(* IEC 61131-3 sources: volt/packages/volt-lsp-iec/test-corpus/pro2193/Device/Plc Logic/Application/09 Misc/Library Manager/L_MC1P_MotionControlBasic (part 5) *)

(* ---- L_MC1P_MOTIONUTILS_I750.pou ---- *)
FUNCTION_BLOCK L_MC1P_MOTIONUTILS_I750 EXTENDS L_MC1P_MotionUtils_Base
VAR
	DRIVETYPE : L_MC1P_DriveType;
	GETAXISEXTENSION : L_MC1P_AxisExtensionTypes;
END_VAR
END_FUNCTION_BLOCK

METHOD GETRETAINMEMINFO : L_MC1P_RetainDataType
VAR_OUTPUT
	MEMINFO : L_MC1P_uAxisRetainInfo;
END_VAR
END_METHOD

(* ---- L_MC1P_MOTIONUTILS_I950.pou ---- *)
FUNCTION_BLOCK L_MC1P_MOTIONUTILS_I950 EXTENDS L_MC1P_MotionUtils_Base
VAR
	DRIVETYPE : L_MC1P_DriveType;
	GETAXISEXTENSION : L_MC1P_AxisExtensionTypes;
END_VAR
END_FUNCTION_BLOCK

METHOD GETRETAINMEMINFO : L_MC1P_RetainDataType
VAR_OUTPUT
	MEMINFO : L_MC1P_uAxisRetainInfo;
END_VAR
END_METHOD

(* ---- L_MC1P_MOTIONUTILS_I950_CIAADV.pou ---- *)
FUNCTION_BLOCK L_MC1P_MOTIONUTILS_I950_CIAADV EXTENDS L_MC1P_MotionUtils_Base
VAR
	DRIVETYPE : L_MC1P_DriveType;
	GETAXISEXTENSION : L_MC1P_AxisExtensionTypes;
END_VAR
END_FUNCTION_BLOCK

METHOD GETRETAINMEMINFO : L_MC1P_RetainDataType
VAR_OUTPUT
	MEMINFO : L_MC1P_uAxisRetainInfo;
END_VAR
END_METHOD

(* ---- L_MC1P_MOTIONUTILS_I950_DRIVE.pou ---- *)
FUNCTION_BLOCK L_MC1P_MOTIONUTILS_I950_DRIVE EXTENDS L_MC1P_MotionUtils_Base
VAR
	DRIVETYPE : L_MC1P_DriveType;
	GETAXISEXTENSION : L_MC1P_AxisExtensionTypes;
END_VAR
END_FUNCTION_BLOCK

METHOD GETGUID : BOOL
VAR_INPUT
	PCONNECTOR : POINTER TO IoConfigConnector;
END_VAR
VAR_IN_OUT
	GUID : L_MC1P_AxisGUID;
END_VAR
END_METHOD

METHOD GETRETAINMEMINFO : L_MC1P_RetainDataType
VAR_OUTPUT
	MEMINFO : L_MC1P_uAxisRetainInfo;
END_VAR
END_METHOD

(* ---- L_MC1P_MOTIONUTILSRETAINHANDLING.pou ---- *)
FUNCTION_BLOCK L_MC1P_MOTIONUTILSRETAINHANDLING
VAR_INPUT
	XRETAINSTART : BOOL;
END_VAR
VAR
	PAXISREAL : POINTER TO _AXIS_REF_REAL;
	PAXISRETAININFORMATION : POINTER TO L_MC1P_AxisRetainInformation;
	RETAININFO : L_MC1P_uAxisRetainInfo;
	ERETAINDATATYPE : L_MC1P_RetainDataType := L_MC1P_RetainDataType.DataRealDrive;
	PRETAINDATA : POINTER TO L_MC1P_uRetainData;
	UINITIALRETAINDATA : L_MC1P_uRetainData;
	XERR_XPOSRECONSTRDATAVERSIONCHANGED : BOOL;
	XERR_POSRECONSTRNODATAAVAILABLE : BOOL;
	XRETAINDATAAVAILABLE : BOOL;
	WRETAINERRORSTATE : WORD;
	WRETAINSTATE : WORD;
	CHECKDRIVEGUID : BOOL;
	DRIVEGUID : L_MC1P_AxisGUID;
	GETAXIS : POINTER TO _Axis_Ref_Real;
	INFO : DWORD;
	ITFRETAINFUNCTION : L_MC1P_IRetainFunction;
	RETAINDATAAVAILABLE : BOOL;
	RETAINDATACONFIGURED : BOOL;
	RETAINSTATE : WORD;
END_VAR
END_FUNCTION_BLOCK

METHOD COPYRETAINDATABYVERSION : BOOL
VAR_INPUT
	PDATA : POINTER TO DWORD;
	INFO : DWORD;
END_VAR
END_METHOD

METHOD GETINITIALDATA : BOOL
VAR_INPUT
	PDATA : POINTER TO DWORD;
	INFO : DWORD;
END_VAR
END_METHOD

METHOD GETINITIALRETAINDATA : POINTER TO L_MC1P_uRetainData
VAR_INPUT
	XNEWEST : BOOL;
END_VAR
END_METHOD

METHOD GETRETAINSTATE : WORD
VAR_OUTPUT
	WSTATERETAINERROR : WORD;
END_VAR
END_METHOD

METHOD REGISTERONRETAINDATAHANDLER
VAR_INPUT
	AXISGUID : L_MC1P_AxisGUID;
END_VAR
END_METHOD

METHOD RESET
END_METHOD

METHOD SETCONNECTEDGUID : BOOL
VAR_INPUT
	GUID : L_MC1P_AxisGUID;
END_VAR
END_METHOD

METHOD SETERRORINFO
VAR_INPUT
	WSTATE : WORD;
END_VAR
END_METHOD

METHOD SETINITIALDATA : BOOL
VAR_INPUT
	PDATA : POINTER TO DWORD;
END_VAR
END_METHOD

METHOD STOREDATA
VAR_INPUT
	PDATA : POINTER TO DWORD;
END_VAR
END_METHOD

METHOD FB_INIT : BOOL
VAR_INPUT
	BINITRETAINS : BOOL;
	BINCOPYCODE : BOOL;
	MEMLENGTH : WORD;
	MEMTYPE : BYTE;
	MEMVERSION : BYTE;
	ERETAINDATATYPE : L_MC1P_RetainDataType;
END_VAR
END_METHOD

(* ---- L_MC1P_MOTIONUTILSRETAINHANDLINGEXTFB.pou ---- *)
FUNCTION_BLOCK L_MC1P_MOTIONUTILSRETAINHANDLINGEXTFB
VAR_INPUT
	XRETAINDATAAVAILABLE : BOOL;
	PRETAINDATA : POINTER TO L_MC1P_uRetainData;
	WRETAINSTATE : WORD;
END_VAR
VAR
	CHECKDRIVEGUID : BOOL;
	DRIVEGUID : L_MC1P_AxisGUID;
	GETAXIS : POINTER TO _Axis_Ref_Real;
	ITFRETAINFUNCTION : L_MC1P_IRetainFunction;
	RETAINDATAAVAILABLE : BOOL;
END_VAR
END_FUNCTION_BLOCK

METHOD GETINITIALRETAINDATA : POINTER TO L_MC1P_uRetainData
VAR_INPUT
	XNEWEST : BOOL;
END_VAR
END_METHOD

METHOD GETRETAINSTATE : WORD
VAR_OUTPUT
	WSTATERETAINERROR : WORD;
END_VAR
END_METHOD

METHOD REGISTERONRETAINDATAHANDLER
VAR_INPUT
	AXISGUID : L_MC1P_AxisGUID;
END_VAR
END_METHOD

METHOD RESET
END_METHOD

METHOD SETCONNECTEDGUID : BOOL
VAR_INPUT
	GUID : L_MC1P_AxisGUID;
END_VAR
END_METHOD

(* ---- L_MC1P_MOTIONUTILSRETAINHANDLINGUNIVERSAL.pou ---- *)
FUNCTION_BLOCK L_MC1P_MOTIONUTILSRETAINHANDLINGUNIVERSAL EXTENDS L_MC1P_MotionUtilsRetainHandling
VAR
	MYDRIVEGUID : L_MC1P_AxisGUID;
	CHECKDRIVEGUID : BOOL;
	DRIVEGUID : L_MC1P_AxisGUID;
END_VAR
END_FUNCTION_BLOCK

METHOD GETINITIALRETAINDATA : POINTER TO L_MC1P_uRetainData
VAR_INPUT
	XNEWEST : BOOL;
END_VAR
END_METHOD

METHOD RESET
END_METHOD

METHOD SETCONNECTEDGUID : BOOL
VAR_INPUT
	GUID : L_MC1P_AxisGUID;
END_VAR
END_METHOD

METHOD STOREDATA
VAR_INPUT
	PDATA : POINTER TO DWORD;
END_VAR
END_METHOD

(* ---- L_MC1P_MOVEABSOLUTE_INERNAL.pou ---- *)
FUNCTION_BLOCK L_MC1P_MOVEABSOLUTE_INERNAL EXTENDS L_MC1P_Template_IntFB
VAR_INPUT
	EXECUTE : BOOL;
	CONTINUOUSUPDATE : BOOL;
	POSITION : LREAL;
	VELOCITY : LREAL;
	ACCELERATION : LREAL;
	DECELERATION : LREAL;
	JERK : LREAL;
	JERKDEC : LREAL;
	DIRECTION : MC_DIRECTION;
	BUFFERMODE : MC_BUFFER_MODE;
END_VAR
VAR_OUTPUT
	DONE : BOOL;
	BUSY : BOOL;
	ACTIVE : BOOL;
	COMMANDABORTED : BOOL;
	ERROR : BOOL;
	ERRORID : L_IE1P_Error;
END_VAR
VAR
	FBMB : L_MC1P_MoveBasic := STRUCT(wCalcProfileMode := 1);
	XUSED : BOOL;
	ABORTEDBYLIMIT : BOOL;
END_VAR
END_FUNCTION_BLOCK

METHOD MAIN
VAR_IN_OUT
	AXIS : AXIS_REF;
	FBBASE : L_MC1P_Template_ForAxis;
END_VAR
END_METHOD

(* ---- L_MC1P_MOVEBASIC.pou ---- *)
FUNCTION_BLOCK L_MC1P_MOVEBASIC
VAR_INPUT
	LRJERKDEC : LREAL := 0;
	XWAIT : BOOL;
	XRECALCULATE : BOOL;
	LRCORRECTTIMEBASE : LREAL;
	WCALCPROFILEMODE : WORD := 0;
	XUSEEXTERNPROFILECALCULATION : BOOL;
	ITFPOSPROFILECALCULATION : L_MC1P_IPosProfileCalculation;
	XENABLEOFFSETVELOCITY : BOOL;
	LROFFSETVELOCITY : LREAL;
	XFINISHPOSFROMMOVEREL : BOOL := FALSE;
END_VAR
VAR
	XSTART : BOOL;
	EXECUTEOLD : BOOL;
	COMMANDABORTEDOLD : BOOL;
	PG : REFERENCE TO L_MC1P_PosProfiler;
	SCPARAM : L_MC1P_ProfileParameter;
	SCPARAMLIM : L_MC1P_ProfileParameter;
	WFUNID : WORD;
	XSETENDVELOCITYBYBUFFERMODE : BOOL;
	XRESETOUTPUT : BOOL;
	EACTSTATE : L_MC1P_AXIS_STATE;
	XCONTINUOUSUPDATEACTIVE : BOOL;
	XSUPERIMPOSED : BOOL;
	XPOSACTIVE : BOOL;
	XVELUPDATE : BOOL;
	XBUFFERACTIVE : BOOL;
	XPOSSWLIMIT : BOOL;
	XNEGSWLIMIT : BOOL;
	XABORTEDBYLIMIT : BOOL;
	XWARNING : BOOL;
	EWARNINGID : L_IE1P_Error;
	XWARNINGOLD : BOOL;
	EWARNINGIDOLD : L_IE1P_Error;
	XLOGINFO : BOOL;
	ELOGINFOID : L_IE1P_Error;
	ELOGINFOIDOLD : L_IE1P_Error;
	XLIMITOLD : BOOL;
	XCONTMODE : BOOL;
	XDONESAVE : BOOL;
	LRPOSLATCHED : LREAL;
	LRPOSSAVE : LREAL;
	XDONEOLD : BOOL;
	LRDISTANCE : LREAL;
	LRSTARTPOS : LREAL;
	LRTMPPOSOFFSET : LREAL;
	XIGNOREMODULOWINDOW : BOOL;
	SCPROFILEDATATMP : L_MC1P_ProfileData;
	SCPROFILEPARATMP : L_MC1P_ProfileParameter;
	XNEWPROFILESTARTAFTERSTANDSTILL : BOOL;
	ESETDIRECTIONMOVEFB : MC_DIRECTION;
	XPOSPROFILERINUSE : BOOL;
	WSTRETCHPROFILEMODE : WORD;
	XBUFFERDATAUPDATED : BOOL;
	XENABLEBUFFER_INT : BOOL;
	SCBUFFERDATA_INT : L_MC1P_BufferData;
	XUPDATEBUFFERDATAFROMDUMMYPG : BOOL;
	PAXIS : POINTER TO AXIS_REF;
	IGNOREMODULOWINDOW : BOOL;
	POSPROFILERINUSE : BOOL;
	PROFILETIME : TIME;
	REMAININGTIMEOFPROFILE : LREAL;
	REMAININGTIMEOFPROFILEAVAILABLE : BOOL;
	STRETCHPROFILEMODE : WORD;
END_VAR
END_FUNCTION_BLOCK

METHOD CALCTARGETPOSITION : LREAL
VAR_INPUT
	POSITION : LREAL;
	DIRECTION : MC_DIRECTION;
	ETRAVERSINGRANGE : L_MC1P_TraversingRange;
	ETYPEFUNCTION : L_MC1P_TypeFunction;
	XFIRSTCALC : BOOL;
	XABORTED : BOOL;
	PROFILEPARAM : L_MC1P_ProfileParameter;
	EAXISSTATEOLD : L_MC1P_AXIS_STATE;
END_VAR
VAR_OUTPUT
	XERROR : BOOL;
	EERRORID : L_IE1P.L_IE1P_Error;
END_VAR
VAR_IN_OUT
	AXIS : AXIS_REF;
END_VAR
END_METHOD

METHOD CHECKDEVIATION : BOOL
VAR_INPUT
	LRINPUT : LREAL;
	LRSAVE : LREAL;
END_VAR
END_METHOD

METHOD CHECKLIMITATION
VAR_INPUT
	EFUNCTIONTYP : L_MC1P_TypeFunction;
	PXPOSMODE : POINTER TO BOOL;
END_VAR
VAR_IN_OUT
	AXIS : AXIS_REF;
	FBBASE : L_MC1P_Template_ForAxis;
	ERROR : BOOL;
	ERRORID : L_IE1P_Error;
END_VAR
END_METHOD

METHOD DETERMINETARGETSPEEDSIGN : BOOL
VAR_INPUT
	LRPOSITION : LREAL;
	ETYPEFUNCTION : L_MC1P_TypeFunction;
	EDIRECTION : MC_DIRECTION;
END_VAR
VAR_IN_OUT
	AXIS : AXIS_REF;
END_VAR
END_METHOD

METHOD INTOLERANCEWINDOW : BOOL
VAR_INPUT
	LRPOSITION : LREAL;
END_VAR
VAR_OUTPUT
	DIRECTION : MC_DIRECTION;
END_VAR
VAR_IN_OUT
	AXIS : AXIS_REF;
END_VAR
END_METHOD

METHOD PREPAREBUFFERDATA
VAR_INPUT
	XENABLEBUFFER : BOOL;
	SCBUFFERDATA : L_MC1P_BufferData;
END_VAR
END_METHOD

METHOD PROFILER : BOOL
VAR_INPUT
	EXECUTE : BOOL;
	CONTINUOUSUPDATE : BOOL;
	POSITION : LREAL;
	VELOCITY : LREAL;
	ENDVELOCITY : LREAL;
	ACCELERATION : LREAL;
	DECELERATION : LREAL;
	JERK : LREAL;
	XPOSMODE : BOOL;
	DIRECTION : MC_DIRECTION;
	BUFFERMODE : MC_BUFFER_MODE;
	EFUNCTIONTYP : L_MC1P_TypeFunction;
END_VAR
VAR_IN_OUT
	AXIS : AXIS_REF;
	DONE : BOOL;
	BUSY : BOOL;
	ACTIVE : BOOL;
	COMMANDABORTED : BOOL;
	ERROR : BOOL;
	ERRORID : L_IE1P_Error;
	FBBASE : L_MC1P_Template_ForAxis;
END_VAR
END_METHOD

METHOD RESET
END_METHOD

METHOD RESETEXECUTE
END_METHOD

(* ---- L_MC1P_MOVERELATIVE_INTERNAL.pou ---- *)
FUNCTION_BLOCK L_MC1P_MOVERELATIVE_INTERNAL EXTENDS L_MC1P_Template_IntFB
VAR_INPUT
	EXECUTE : BOOL;
	CONTINUOUSUPDATE : BOOL;
	DISTANCE : LREAL;
	VELOCITY : LREAL;
	ACCELERATION : LREAL;
	DECELERATION : LREAL;
	JERK : LREAL;
	JERKDEC : LREAL;
	BUFFERMODE : MC_BUFFER_MODE;
	XUSEEXTERNPROFILECALCULATION : BOOL;
	ITFPOSPROFILECALCULATION : L_MC1P_IPosProfileCalculation;
END_VAR
VAR_OUTPUT
	DONE : BOOL;
	BUSY : BOOL;
	ACTIVE : BOOL;
	COMMANDABORTED : BOOL;
	ERROR : BOOL;
	ERRORID : L_IE1P_Error;
END_VAR
VAR
	FBMB : L_MC1P_MoveBasic := STRUCT(wCalcProfileMode := 1);
	XUSED : BOOL;
	ABORTEDBYLIMIT : BOOL;
END_VAR
END_FUNCTION_BLOCK

METHOD MAIN
VAR_IN_OUT
	AXIS : AXIS_REF;
	FBBASE : L_MC1P_Template_ForAxis;
END_VAR
END_METHOD

(* ---- L_MC1P_MOVEVELOCITY_INTERNAL.pou ---- *)
FUNCTION_BLOCK L_MC1P_MOVEVELOCITY_INTERNAL EXTENDS L_MC1P_Template_IntFB
VAR_INPUT
	EXECUTE : BOOL;
	CONTINUOUSUPDATE : BOOL;
	VELOCITY : LREAL;
	ACCELERATION : LREAL;
	DECELERATION : LREAL;
	JERK : LREAL;
	JERKDEC : LREAL;
	DIRECTION : MC_DIRECTION := MC_DIRECTION.mcPositiveDirection;
	BUFFERMODE : MC_BUFFER_MODE;
	XUSEEXTERNPROFILECALCULATION : BOOL;
	ITFPOSPROFILECALCULATION : L_MC1P_IPosProfileCalculation;
	XENABLEOFFSETVELOCITY : BOOL;
	LROFFSETVELOCITY : LREAL;
END_VAR
VAR_OUTPUT
	INVELOCITY : BOOL;
	BUSY : BOOL;
	ACTIVE : BOOL;
	COMMANDABORTED : BOOL;
	ERROR : BOOL;
	ERRORID : L_IE1P_Error;
END_VAR
VAR
	FBMB : L_MC1P_MoveBasic := STRUCT(wCalcProfileMode := 1);
	LRVEL : LREAL;
	XUSED : BOOL;
	ABORTEDBYLIMIT : BOOL;
END_VAR
END_FUNCTION_BLOCK

METHOD MAIN
VAR_IN_OUT
	AXIS : AXIS_REF;
	FBBASE : L_MC1P_Template_ForAxis;
END_VAR
END_METHOD

METHOD MODVELOCITY : LREAL
VAR_IN_OUT
	AXIS : AXIS_REF;
END_VAR
END_METHOD

(* ---- L_MC1P_MPOT.pou ---- *)
FUNCTION_BLOCK L_MC1P_MPOT
VAR_INPUT
	XENABLE : BOOL;
	XJOGPOS : BOOL;
	XJOGNEG : BOOL;
	LRVELPOS : LREAL;
	LRVELNEG : LREAL;
	LRACC : LREAL;
	LRDEC : LREAL;
	LRDECDISABLE : LREAL;
END_VAR
VAR_OUTPUT
	XBUSY : BOOL;
	LRSETVELOUT : LREAL;
END_VAR
VAR
	HLP_MPOT : L_MC1P_HlpRampGenerator;
	XJOGPOSITIVEFLAG : BOOL;
	XJOGNEGATIVEFLAG : BOOL;
END_VAR
END_FUNCTION_BLOCK

(* ---- L_MC1P_NOISEDETECTION.pou ---- *)
FUNCTION_BLOCK L_MC1P_NOISEDETECTION
VAR_INPUT
	XENABLE : BOOL;
	LRCYCPOS : LREAL;
	LRCYCVEL : LREAL;
	LRCYCACC : LREAL;
	ECYCVALUEMODE : L_MC1P_SetValueMode := L_MC1P_SetValueMode.Vel;
	LRCYCLELENGTH : LREAL := 360;
	ETRAVERSINGRANGE : L_MC1P_TraversingRange;
END_VAR
VAR_OUTPUT
	XBUSY : BOOL;
	XNOISEDETECTED : BOOL;
END_VAR
VAR
	WSTATE : WORD;
	XNOISE_INT : BOOL;
	LRDELTAPOS_INT : LREAL;
	WNOISEDETECTEDCOUNT : WORD;
	WNOISENOTDETECTEDCOUNT : WORD;
	XENABLE_OLD : BOOL;
	LRCYCPOS_OLD : LREAL;
	LRCYCVEL_OLD : LREAL;
	LRDELTAPOS_OLD : LREAL;
	FB_STACK : L_MC1P_StackControlArray := STRUCT(iMaxLegth := ciArraylengthAtCheckNoise);
	ALRACC : ARRAY [1..ciArraylengthAtCheckNoise] OF LREAL;
	ALRDELTA2POS : ARRAY [1..ciArraylengthAtCheckNoise] OF LREAL;
	ALRDELTAVEL : ARRAY [1..ciArraylengthAtCheckNoise] OF LREAL;
	CIARRAYLENGTHATCHECKNOISE : INT := 15;
	C_WHYSTCOUNTERNOISEDETECTED : WORD := 3;
END_VAR
END_FUNCTION_BLOCK

METHOD CALL_ERRORHANDLER
END_METHOD

METHOD CALL_FBMETHODS
END_METHOD

METHOD CALL_OUTPUT
END_METHOD

METHOD CALL_RESETCOMMANDS
END_METHOD

METHOD CALL_RESETOUTPUT
END_METHOD

METHOD CALL_STATEMACHINE
END_METHOD

METHOD FUN_CHECKARRAY : BOOL
VAR_INPUT
	ISTACKSTARTPOS : INT;
	ISTACKLENGTH : INT;
END_VAR
VAR_IN_OUT
	ALRVALUE : ARRAY [1..ciArraylengthAtCheckNoise] OF LREAL;
END_VAR
END_METHOD

METHOD FUN_CHECKARRAY2 : BOOL
VAR_INPUT
	ISTACKSTARTPOS : INT;
	ISTACKLENGTH : INT;
END_VAR
VAR_IN_OUT
	ALRVALUE1 : ARRAY [1..ciArraylengthAtCheckNoise] OF LREAL;
	ALRVALUE2 : ARRAY [1..ciArraylengthAtCheckNoise] OF LREAL;
END_VAR
END_METHOD

METHOD FUN_CHECKARRAY3 : BOOL
VAR_INPUT
	ISTACKSTARTPOS : INT;
	ISTACKLENGTH : INT;
END_VAR
VAR_IN_OUT
	ALRVALUE1 : ARRAY [1..ciArraylengthAtCheckNoise] OF LREAL;
	ALRVALUE2 : ARRAY [1..ciArraylengthAtCheckNoise] OF LREAL;
	ALRVALUE3 : ARRAY [1..ciArraylengthAtCheckNoise] OF LREAL;
END_VAR
END_METHOD

METHOD FUN_CHECKNOISE : BOOL
VAR_IN_OUT
	LRVALUE1 : LREAL;
	LRVALUE2 : LREAL;
	LRVALUE3 : LREAL;
	LRVALUE4 : LREAL;
	INOTMONOTONCOUNTER : INT;
END_VAR
END_METHOD

METHOD CALL_INIT
END_METHOD

(* ---- L_MC1P_OFFSETGENERATOR.pou ---- *)
FUNCTION_BLOCK L_MC1P_OFFSETGENERATOR
VAR_INPUT
	XENABLE : BOOL;
	LRCYCMASTERPOS : LREAL;
	LRCYCMASTERVEL : LREAL;
	LRCYCMASTERACC : LREAL;
	LRSETOFFSET : LREAL;
	XLOADOFFSET : BOOL;
	DWNUMERATOR : DWORD := 1;
	DWDENOMINATOR : DWORD := 1;
	EDIRECTION : L_MC1P_Direction;
	EPROFILETYPE : L_MC1P_ProfileType := 0;
	LRVELPOS : LREAL := 100.0;
	LRVELNEG : LREAL := 100.0;
	LRACCDEC : LREAL := 1000.0;
END_VAR
VAR_OUTPUT
	XBUSY : BOOL;
	XDONE : BOOL;
	LROFFSET : LREAL;
	LRSETOFFSETVELOUT : LREAL;
END_VAR
VAR_IN_OUT
	MASTERAXIS : AXIS_REF;
	SLAVEAXIS : AXIS_REF;
END_VAR
VAR
	WSTATEMASHINESIMPLEPOS : WORD := 0;
	LRSMDELTAPOS : LREAL;
	LRSIMPLEPOSOFFSET : LREAL;
	LRSALVEVELBAND : LREAL;
	LRABORTSTARTVEL : LREAL;
	LRSMSETOFFSET_OLD : LREAL;
	LRFACTOR : LREAL;
	LRLOADRESTOFFSET_INT : LREAL;
	XENABLE_OLD : BOOL;
	LROFFSET_OLD : LREAL;
	SIMPLEPOSITIONING : L_MC1P_PosGenerator;
	ABORTPOSCTRLCORRECT : L_MC1P_PosGeneratorAbortCorrection;
END_VAR
END_FUNCTION_BLOCK

METHOD CALL_CALCFACTOR
END_METHOD

METHOD CALL_ERRORHANDLER
END_METHOD

METHOD CALL_FBMETHODS
END_METHOD

METHOD CALL_OUTPUT
END_METHOD

METHOD CALL_RESETCOMMANDS
END_METHOD

METHOD CALL_RESETOUTPUT
END_METHOD

METHOD CALL_SIMPLEPOS
END_METHOD

METHOD CALL_SIMPLEPOS_ABORTPOSCTRLCORRECT
END_METHOD

METHOD CALL_SIMPLEPOS_OFFSET
END_METHOD

METHOD CALL_STATEMASHINE
END_METHOD

(* ---- L_MC1P_OPTICALTRACKING.pou ---- *)
FUNCTION_BLOCK L_MC1P_OPTICALTRACKING EXTENDS L_MC1P_Template
VAR_INPUT
	XEXECUTE : BOOL := FALSE;
	RTIME : REAL := 5.0;
END_VAR
VAR_OUTPUT
	XDONE : BOOL := FALSE;
	XBUSY : BOOL;
	XERROR : BOOL;
	EERRORID : L_IE1P_Error;
END_VAR
VAR
	XEXECUTEOLD : BOOL := FALSE;
	XVALID : BOOL := FALSE;
	XACTIV : BOOL := FALSE;
	XBUSYINT : BOOL := FALSE;
	XDONEINT : BOOL := FALSE;
	WSTATE : WORD;
	DWPARLENGTH : DWORD := 2;
	WPARAMNUMBER : WORD := 16#2021;
	BYSUBCODE : BYTE := 1;
	DNVALUE : DINT;
	WP : MC_WriteParameter;
	RP : MC_ReadParameter;
END_VAR
END_FUNCTION_BLOCK

(* ---- L_MC1P_OPTIMIZEPOSQUANTISATION.pou ---- *)
FUNCTION_BLOCK L_MC1P_OPTIMIZEPOSQUANTISATION
VAR_INPUT
	DINEWPOSIN : DINT;
	LRTIMEDIFFTOLASTPOS : LREAL;
	LRTIMEDIFFAPPSTART : LREAL;
END_VAR
VAR_OUTPUT
	LRNEWENCODERPOS : LREAL;
	DINEWENCODERPOS : DINT;
	LRRESIDUAL : LREAL;
	XUPDATETPDATA : BOOL;
END_VAR
VAR_IN_OUT
	AXIS : _AXIS_REF_REAL;
END_VAR
VAR
	DIOLDPOS : DINT;
	WCOUNTER : WORD;
	WUPDATECYCLE : WORD;
	WLASTUPDATECYCLE : WORD;
	WCYCLEDIFF : LREAL;
	LRPOSDIFF : LREAL;
	WCNTIDX : WORD;
	AWSAMPLECOUNTER : ARRAY [0..7] OF LREAL;
	ADINEWPOSDIFF : ARRAY [0..7] OF DINT;
	WVALIDVALUES : WORD := 0;
	LROLDENCPOS : LREAL;
	LRFACTOR : LREAL;
	DIDIRECTION : DINT;
	WMAXVALIDVALUES : WORD := 2;
	LROLDENCODERPOS : LREAL;
	IDX : WORD;
	DIMAXDIRECTIONCNT : DINT := 6;
	LRTMP : LREAL;
	WCOUNTEROLD : WORD;
	LROLDTPPOS : LREAL;
	LRNEWTPPOS : LREAL;
	WTPCYCLEDIFF : WORD;
	XDEBUG : BOOL;
END_VAR
END_FUNCTION_BLOCK

METHOD GETPOSDIFF : LREAL
END_METHOD

METHOD GETPOSDIFFDINTRANGE : LREAL
VAR_INPUT
	LRPOS1 : LREAL;
	LRPOS2 : LREAL;
END_VAR
END_METHOD

METHOD GETVELOCITY : LREAL
VAR_INPUT
	DWTASKYCLE_US : DWORD;
END_VAR
END_METHOD

METHOD OPTIMIZETPTIMESTAMPS : BOOL
VAR_INPUT
	XACTIVATERAWPOSHANDLING : BOOL;
END_VAR
VAR_IN_OUT
	AXIS : _AXIS_REF_REAL;
END_VAR
END_METHOD

METHOD POSTODINTRANGE : LREAL
VAR_INPUT
	LRPOS : LREAL;
END_VAR
END_METHOD

METHOD RESET : BOOL
VAR_INPUT
	DIINITPOS : DINT;
END_VAR
END_METHOD

(* ---- L_MC1P_PARAINTERFACE_AXIS_REF_9400HL.pou ---- *)
FUNCTION_BLOCK L_MC1P_PARAINTERFACE_AXIS_REF_9400HL
VAR
	ASCVALUERANGES : ARRAY [0..5] OF L_MC1P_MinMaxValue;
END_VAR
END_FUNCTION_BLOCK

METHOD HLP_READBOOLPARAMETER : BOOL
VAR_INPUT
	PINPUTDATA : POINTER TO BYTE;
	PARAMETER : DINT;
	PXVALUE : POINTER TO BOOL;
	XALLOWINVISIBLE : BOOL;
END_VAR
END_METHOD

METHOD HLP_READPARAMETER : BOOL
VAR_INPUT
	PINPUTDATA : POINTER TO BYTE;
	PARAMETER : DINT;
	PLRVALUE : POINTER TO LREAL;
	XALLOWINVISIBLE : BOOL;
END_VAR
END_METHOD

METHOD HLP_WRITEBOOLPARAMETER : BOOL
VAR_INPUT
	PINPUTDATA : POINTER TO BYTE;
	PARAMETER : DINT;
	PXVALUE : POINTER TO BOOL;
	XALLOWINVISIBLE : BOOL;
END_VAR
VAR_OUTPUT
	WERRORID : WORD;
END_VAR
END_METHOD

METHOD HLP_WRITEPARAMETER : BOOL
VAR_INPUT
	PINPUTDATA : POINTER TO BYTE;
	PARAMETER : DINT;
	PLRVALUE : POINTER TO LREAL;
	XALLOWINVISIBLE : BOOL;
END_VAR
VAR_OUTPUT
	WERRORID : WORD;
END_VAR
END_METHOD

METHOD HLP_INITPARREF : BOOL
VAR_INPUT
	PINPUTDATA : POINTER TO BYTE;
	PINPUTDATA2 : POINTER TO BYTE;
END_VAR
VAR_OUTPUT
	WERRORID : WORD;
END_VAR
END_METHOD

METHOD HLP_GETPARAMETERPROPERTIES : BOOL
VAR_INPUT
	PAXISREF : POINTER TO AXIS_REF;
	DIPARAMETER : DINT;
	XALLOWINVISIBLE : BOOL;
END_VAR
VAR_OUTPUT
	PPARAMADDR : POINTER TO BYTE := 0;
	EORDINALTYPE : L_MC1P_OrdinalType := L_MC1P_OrdinalType.otNONE;
	XREADWRITE : BOOL := FALSE;
	LRUNITFACTOR : LREAL := 0.0;
	LRDEFAULTVALUE : LREAL := 0.0;
	WVALUERANGES : WORD := 0;
	PVALUERANGES : POINTER TO L_MC1P_MinMaxValue := 0;
END_VAR
END_METHOD

(* ---- L_MC1P_PARAINTERFACE_AXIS_REF_9400HL_CAN.pou ---- *)
FUNCTION_BLOCK L_MC1P_PARAINTERFACE_AXIS_REF_9400HL_CAN
VAR
	ASCVALUERANGES : ARRAY [0..5] OF L_MC1P_MinMaxValue;
END_VAR
END_FUNCTION_BLOCK

METHOD HLP_READBOOLPARAMETER : BOOL
VAR_INPUT
	PINPUTDATA : POINTER TO BYTE;
	PARAMETER : DINT;
	PXVALUE : POINTER TO BOOL;
	XALLOWINVISIBLE : BOOL;
END_VAR
END_METHOD

METHOD HLP_READPARAMETER : BOOL
VAR_INPUT
	PINPUTDATA : POINTER TO BYTE;
	PARAMETER : DINT;
	PLRVALUE : POINTER TO LREAL;
	XALLOWINVISIBLE : BOOL;
END_VAR
END_METHOD

METHOD HLP_WRITEBOOLPARAMETER : BOOL
VAR_INPUT
	PINPUTDATA : POINTER TO BYTE;
	PARAMETER : DINT;
	PXVALUE : POINTER TO BOOL;
	XALLOWINVISIBLE : BOOL;
END_VAR
VAR_OUTPUT
	WERRORID : WORD;
END_VAR
END_METHOD

METHOD HLP_WRITEPARAMETER : BOOL
VAR_INPUT
	PINPUTDATA : POINTER TO BYTE;
	PARAMETER : DINT;
	PLRVALUE : POINTER TO LREAL;
	XALLOWINVISIBLE : BOOL;
END_VAR
VAR_OUTPUT
	WERRORID : WORD;
END_VAR
END_METHOD

METHOD HLP_INITPARREF : BOOL
VAR_INPUT
	PINPUTDATA : POINTER TO BYTE;
	PINPUTDATA2 : POINTER TO BYTE;
END_VAR
VAR_OUTPUT
	WERRORID : WORD;
END_VAR
END_METHOD

METHOD HLP_GETPARAMETERPROPERTIES : BOOL
VAR_INPUT
	PAXISREF : POINTER TO AXIS_REF;
	DIPARAMETER : DINT;
	XALLOWINVISIBLE : BOOL;
END_VAR
VAR_OUTPUT
	PPARAMADDR : POINTER TO BYTE := 0;
	EORDINALTYPE : L_MC1P_OrdinalType := L_MC1P_OrdinalType.otNONE;
	XREADWRITE : BOOL := FALSE;
	LRUNITFACTOR : LREAL := 0.0;
	LRDEFAULTVALUE : LREAL := 0.0;
	WVALUERANGES : WORD := 0;
	PVALUERANGES : POINTER TO L_MC1P_MinMaxValue := 0;
END_VAR
END_METHOD

(* ---- L_MC1P_PARAINTERFACE_AXIS_REF_ENC_BPB.pou ---- *)
FUNCTION_BLOCK L_MC1P_PARAINTERFACE_AXIS_REF_ENC_BPB
VAR
	ASCVALUERANGES : ARRAY [0..22] OF L_MC1P_MinMaxValue;
END_VAR
END_FUNCTION_BLOCK

METHOD HLP_READBOOLPARAMETER : BOOL
VAR_INPUT
	PINPUTDATA : POINTER TO BYTE;
	PARAMETER : DINT;
	PXVALUE : POINTER TO BOOL;
	XALLOWINVISIBLE : BOOL;
END_VAR
END_METHOD

METHOD HLP_READPARAMETER : BOOL
VAR_INPUT
	PINPUTDATA : POINTER TO BYTE;
	PARAMETER : DINT;
	PLRVALUE : POINTER TO LREAL;
	XALLOWINVISIBLE : BOOL;
END_VAR
END_METHOD

METHOD HLP_WRITEBOOLPARAMETER : BOOL
VAR_INPUT
	PINPUTDATA : POINTER TO BYTE;
	PARAMETER : DINT;
	PXVALUE : POINTER TO BOOL;
	XALLOWINVISIBLE : BOOL;
END_VAR
VAR_OUTPUT
	WERRORID : WORD;
END_VAR
END_METHOD

METHOD HLP_WRITEPARAMETER : BOOL
VAR_INPUT
	PINPUTDATA : POINTER TO BYTE;
	PARAMETER : DINT;
	PLRVALUE : POINTER TO LREAL;
	XALLOWINVISIBLE : BOOL;
END_VAR
VAR_OUTPUT
	WERRORID : WORD;
END_VAR
END_METHOD

METHOD HLP_INITPARREF : BOOL
VAR_INPUT
	PINPUTDATA : POINTER TO BYTE;
	PINPUTDATA2 : POINTER TO BYTE;
END_VAR
VAR_OUTPUT
	WERRORID : WORD;
END_VAR
END_METHOD

METHOD HLP_GETPARAMETERPROPERTIES : BOOL
VAR_INPUT
	PAXISREF : POINTER TO AXIS_REF;
	DIPARAMETER : DINT;
	XALLOWINVISIBLE : BOOL;
END_VAR
VAR_OUTPUT
	PPARAMADDR : POINTER TO BYTE := 0;
	EORDINALTYPE : L_MC1P_OrdinalType := L_MC1P_OrdinalType.otNONE;
	XREADWRITE : BOOL := FALSE;
	LRUNITFACTOR : LREAL := 0.0;
	LRDEFAULTVALUE : LREAL := 0.0;
	WVALUERANGES : WORD := 0;
	PVALUERANGES : POINTER TO L_MC1P_MinMaxValue := 0;
END_VAR
END_METHOD

(* ---- L_MC1P_PARAINTERFACE_AXIS_REF_ENC_FREE.pou ---- *)
FUNCTION_BLOCK L_MC1P_PARAINTERFACE_AXIS_REF_ENC_FREE
VAR
	ASCVALUERANGES : ARRAY [0..22] OF L_MC1P_MinMaxValue;
END_VAR
END_FUNCTION_BLOCK

METHOD HLP_READBOOLPARAMETER : BOOL
VAR_INPUT
	PINPUTDATA : POINTER TO BYTE;
	PARAMETER : DINT;
	PXVALUE : POINTER TO BOOL;
	XALLOWINVISIBLE : BOOL;
END_VAR
END_METHOD

METHOD HLP_READPARAMETER : BOOL
VAR_INPUT
	PINPUTDATA : POINTER TO BYTE;
	PARAMETER : DINT;
	PLRVALUE : POINTER TO LREAL;
	XALLOWINVISIBLE : BOOL;
END_VAR
END_METHOD

METHOD HLP_WRITEBOOLPARAMETER : BOOL
VAR_INPUT
	PINPUTDATA : POINTER TO BYTE;
	PARAMETER : DINT;
	PXVALUE : POINTER TO BOOL;
	XALLOWINVISIBLE : BOOL;
END_VAR
VAR_OUTPUT
	WERRORID : WORD;
END_VAR
END_METHOD

METHOD HLP_WRITEPARAMETER : BOOL
VAR_INPUT
	PINPUTDATA : POINTER TO BYTE;
	PARAMETER : DINT;
	PLRVALUE : POINTER TO LREAL;
	XALLOWINVISIBLE : BOOL;
END_VAR
VAR_OUTPUT
	WERRORID : WORD;
END_VAR
END_METHOD

METHOD HLP_INITPARREF : BOOL
VAR_INPUT
	PINPUTDATA : POINTER TO BYTE;
	PINPUTDATA2 : POINTER TO BYTE;
END_VAR
VAR_OUTPUT
	WERRORID : WORD;
END_VAR
END_METHOD

METHOD HLP_GETPARAMETERPROPERTIES : BOOL
VAR_INPUT
	PAXISREF : POINTER TO AXIS_REF;
	DIPARAMETER : DINT;
	XALLOWINVISIBLE : BOOL;
END_VAR
VAR_OUTPUT
	PPARAMADDR : POINTER TO BYTE := 0;
	EORDINALTYPE : L_MC1P_OrdinalType := L_MC1P_OrdinalType.otNONE;
	XREADWRITE : BOOL := FALSE;
	LRUNITFACTOR : LREAL := 0.0;
	LRDEFAULTVALUE : LREAL := 0.0;
	WVALUERANGES : WORD := 0;
	PVALUERANGES : POINTER TO L_MC1P_MinMaxValue := 0;
END_VAR
END_METHOD

(* ---- L_MC1P_PARAINTERFACE_AXIS_REF_ENC_I500_ECAT.pou ---- *)
FUNCTION_BLOCK L_MC1P_PARAINTERFACE_AXIS_REF_ENC_I500_ECAT
VAR
	ASCVALUERANGES : ARRAY [0..22] OF L_MC1P_MinMaxValue;
END_VAR
END_FUNCTION_BLOCK

METHOD HLP_READBOOLPARAMETER : BOOL
VAR_INPUT
	PINPUTDATA : POINTER TO BYTE;
	PARAMETER : DINT;
	PXVALUE : POINTER TO BOOL;
	XALLOWINVISIBLE : BOOL;
END_VAR
END_METHOD

METHOD HLP_READPARAMETER : BOOL
VAR_INPUT
	PINPUTDATA : POINTER TO BYTE;
	PARAMETER : DINT;
	PLRVALUE : POINTER TO LREAL;
	XALLOWINVISIBLE : BOOL;
END_VAR
END_METHOD

METHOD HLP_WRITEBOOLPARAMETER : BOOL
VAR_INPUT
	PINPUTDATA : POINTER TO BYTE;
	PARAMETER : DINT;
	PXVALUE : POINTER TO BOOL;
	XALLOWINVISIBLE : BOOL;
END_VAR
VAR_OUTPUT
	WERRORID : WORD;
END_VAR
END_METHOD

METHOD HLP_WRITEPARAMETER : BOOL
VAR_INPUT
	PINPUTDATA : POINTER TO BYTE;
	PARAMETER : DINT;
	PLRVALUE : POINTER TO LREAL;
	XALLOWINVISIBLE : BOOL;
END_VAR
VAR_OUTPUT
	WERRORID : WORD;
END_VAR
END_METHOD

METHOD HLP_INITPARREF : BOOL
VAR_INPUT
	PINPUTDATA : POINTER TO BYTE;
	PINPUTDATA2 : POINTER TO BYTE;
END_VAR
VAR_OUTPUT
	WERRORID : WORD;
END_VAR
END_METHOD

METHOD HLP_GETPARAMETERPROPERTIES : BOOL
VAR_INPUT
	PAXISREF : POINTER TO AXIS_REF;
	DIPARAMETER : DINT;
	XALLOWINVISIBLE : BOOL;
END_VAR
VAR_OUTPUT
	PPARAMADDR : POINTER TO BYTE := 0;
	EORDINALTYPE : L_MC1P_OrdinalType := L_MC1P_OrdinalType.otNONE;
	XREADWRITE : BOOL := FALSE;
	LRUNITFACTOR : LREAL := 0.0;
	LRDEFAULTVALUE : LREAL := 0.0;
	WVALUERANGES : WORD := 0;
	PVALUERANGES : POINTER TO L_MC1P_MinMaxValue := 0;
END_VAR
END_METHOD

(* ---- L_MC1P_PARAINTERFACE_AXIS_REF_ENC_I900_DRIVE.pou ---- *)
FUNCTION_BLOCK L_MC1P_PARAINTERFACE_AXIS_REF_ENC_I900_DRIVE
VAR
	ASCVALUERANGES : ARRAY [0..1] OF L_MC1P_MinMaxValue;
END_VAR
END_FUNCTION_BLOCK

METHOD HLP_READBOOLPARAMETER : BOOL
VAR_INPUT
	PINPUTDATA : POINTER TO BYTE;
	PARAMETER : DINT;
	PXVALUE : POINTER TO BOOL;
	XALLOWINVISIBLE : BOOL;
END_VAR
END_METHOD

METHOD HLP_READPARAMETER : BOOL
VAR_INPUT
	PINPUTDATA : POINTER TO BYTE;
	PARAMETER : DINT;
	PLRVALUE : POINTER TO LREAL;
	XALLOWINVISIBLE : BOOL;
END_VAR
END_METHOD

METHOD HLP_WRITEBOOLPARAMETER : BOOL
VAR_INPUT
	PINPUTDATA : POINTER TO BYTE;
	PARAMETER : DINT;
	PXVALUE : POINTER TO BOOL;
	XALLOWINVISIBLE : BOOL;
END_VAR
VAR_OUTPUT
	WERRORID : WORD;
END_VAR
END_METHOD

METHOD HLP_WRITEPARAMETER : BOOL
VAR_INPUT
	PINPUTDATA : POINTER TO BYTE;
	PARAMETER : DINT;
	PLRVALUE : POINTER TO LREAL;
	XALLOWINVISIBLE : BOOL;
END_VAR
VAR_OUTPUT
	WERRORID : WORD;
END_VAR
END_METHOD

METHOD HLP_INITPARREF : BOOL
VAR_INPUT
	PINPUTDATA : POINTER TO BYTE;
	PINPUTDATA2 : POINTER TO BYTE;
END_VAR
VAR_OUTPUT
	WERRORID : WORD;
END_VAR
END_METHOD

METHOD HLP_GETPARAMETERPROPERTIES : BOOL
VAR_INPUT
	PAXISREF : POINTER TO AXIS_REF;
	DIPARAMETER : DINT;
	XALLOWINVISIBLE : BOOL;
END_VAR
VAR_OUTPUT
	PPARAMADDR : POINTER TO BYTE := 0;
	EORDINALTYPE : L_MC1P_OrdinalType := L_MC1P_OrdinalType.otNONE;
	XREADWRITE : BOOL := FALSE;
	LRUNITFACTOR : LREAL := 0.0;
	LRDEFAULTVALUE : LREAL := 0.0;
	WVALUERANGES : WORD := 0;
	PVALUERANGES : POINTER TO L_MC1P_MinMaxValue := 0;
END_VAR
END_METHOD

(* ---- L_MC1P_PARAINTERFACE_AXIS_REF_ENC_I900_DRIVE_CIA.pou ---- *)
FUNCTION_BLOCK L_MC1P_PARAINTERFACE_AXIS_REF_ENC_I900_DRIVE_CIA
VAR
	ASCVALUERANGES : ARRAY [0..1] OF L_MC1P_MinMaxValue;
END_VAR
END_FUNCTION_BLOCK

METHOD HLP_READBOOLPARAMETER : BOOL
VAR_INPUT
	PINPUTDATA : POINTER TO BYTE;
	PARAMETER : DINT;
	PXVALUE : POINTER TO BOOL;
	XALLOWINVISIBLE : BOOL;
END_VAR
END_METHOD

METHOD HLP_READPARAMETER : BOOL
VAR_INPUT
	PINPUTDATA : POINTER TO BYTE;
	PARAMETER : DINT;
	PLRVALUE : POINTER TO LREAL;
	XALLOWINVISIBLE : BOOL;
END_VAR
END_METHOD

METHOD HLP_WRITEBOOLPARAMETER : BOOL
VAR_INPUT
	PINPUTDATA : POINTER TO BYTE;
	PARAMETER : DINT;
	PXVALUE : POINTER TO BOOL;
	XALLOWINVISIBLE : BOOL;
END_VAR
VAR_OUTPUT
	WERRORID : WORD;
END_VAR
END_METHOD

METHOD HLP_WRITEPARAMETER : BOOL
VAR_INPUT
	PINPUTDATA : POINTER TO BYTE;
	PARAMETER : DINT;
	PLRVALUE : POINTER TO LREAL;
	XALLOWINVISIBLE : BOOL;
END_VAR
VAR_OUTPUT
	WERRORID : WORD;
END_VAR
END_METHOD

METHOD HLP_INITPARREF : BOOL
VAR_INPUT
	PINPUTDATA : POINTER TO BYTE;
	PINPUTDATA2 : POINTER TO BYTE;
END_VAR
VAR_OUTPUT
	WERRORID : WORD;
END_VAR
END_METHOD

METHOD HLP_GETPARAMETERPROPERTIES : BOOL
VAR_INPUT
	PAXISREF : POINTER TO AXIS_REF;
	DIPARAMETER : DINT;
	XALLOWINVISIBLE : BOOL;
END_VAR
VAR_OUTPUT
	PPARAMADDR : POINTER TO BYTE := 0;
	EORDINALTYPE : L_MC1P_OrdinalType := L_MC1P_OrdinalType.otNONE;
	XREADWRITE : BOOL := FALSE;
	LRUNITFACTOR : LREAL := 0.0;
	LRDEFAULTVALUE : LREAL := 0.0;
	WVALUERANGES : WORD := 0;
	PVALUERANGES : POINTER TO L_MC1P_MinMaxValue := 0;
END_VAR
END_METHOD

(* ---- L_MC1P_PARAINTERFACE_AXIS_REF_ENC_I900_ECAT.pou ---- *)
FUNCTION_BLOCK L_MC1P_PARAINTERFACE_AXIS_REF_ENC_I900_ECAT
VAR
	ASCVALUERANGES : ARRAY [0..7] OF L_MC1P_MinMaxValue;
END_VAR
END_FUNCTION_BLOCK

METHOD HLP_READBOOLPARAMETER : BOOL
VAR_INPUT
	PINPUTDATA : POINTER TO BYTE;
	PARAMETER : DINT;
	PXVALUE : POINTER TO BOOL;
	XALLOWINVISIBLE : BOOL;
END_VAR
END_METHOD

METHOD HLP_READPARAMETER : BOOL
VAR_INPUT
	PINPUTDATA : POINTER TO BYTE;
	PARAMETER : DINT;
	PLRVALUE : POINTER TO LREAL;
	XALLOWINVISIBLE : BOOL;
END_VAR
END_METHOD

METHOD HLP_WRITEBOOLPARAMETER : BOOL
VAR_INPUT
	PINPUTDATA : POINTER TO BYTE;
	PARAMETER : DINT;
	PXVALUE : POINTER TO BOOL;
	XALLOWINVISIBLE : BOOL;
END_VAR
VAR_OUTPUT
	WERRORID : WORD;
END_VAR
END_METHOD

METHOD HLP_WRITEPARAMETER : BOOL
VAR_INPUT
	PINPUTDATA : POINTER TO BYTE;
	PARAMETER : DINT;
	PLRVALUE : POINTER TO LREAL;
	XALLOWINVISIBLE : BOOL;
END_VAR
VAR_OUTPUT
	WERRORID : WORD;
END_VAR
END_METHOD

METHOD HLP_INITPARREF : BOOL
VAR_INPUT
	PINPUTDATA : POINTER TO BYTE;
	PINPUTDATA2 : POINTER TO BYTE;
END_VAR
VAR_OUTPUT
	WERRORID : WORD;
END_VAR
END_METHOD

METHOD HLP_GETPARAMETERPROPERTIES : BOOL
VAR_INPUT
	PAXISREF : POINTER TO AXIS_REF;
	DIPARAMETER : DINT;
	XALLOWINVISIBLE : BOOL;
END_VAR
VAR_OUTPUT
	PPARAMADDR : POINTER TO BYTE := 0;
	EORDINALTYPE : L_MC1P_OrdinalType := L_MC1P_OrdinalType.otNONE;
	XREADWRITE : BOOL := FALSE;
	LRUNITFACTOR : LREAL := 0.0;
	LRDEFAULTVALUE : LREAL := 0.0;
	WVALUERANGES : WORD := 0;
	PVALUERANGES : POINTER TO L_MC1P_MinMaxValue := 0;
END_VAR
END_METHOD

(* ---- L_MC1P_PARAINTERFACE_AXIS_REF_ENC_IO_ETC.pou ---- *)
FUNCTION_BLOCK L_MC1P_PARAINTERFACE_AXIS_REF_ENC_IO_ETC
VAR
	ASCVALUERANGES : ARRAY [0..22] OF L_MC1P_MinMaxValue;
END_VAR
END_FUNCTION_BLOCK

METHOD HLP_READBOOLPARAMETER : BOOL
VAR_INPUT
	PINPUTDATA : POINTER TO BYTE;
	PARAMETER : DINT;
	PXVALUE : POINTER TO BOOL;
	XALLOWINVISIBLE : BOOL;
END_VAR
END_METHOD

METHOD HLP_READPARAMETER : BOOL
VAR_INPUT
	PINPUTDATA : POINTER TO BYTE;
	PARAMETER : DINT;
	PLRVALUE : POINTER TO LREAL;
	XALLOWINVISIBLE : BOOL;
END_VAR
END_METHOD

METHOD HLP_WRITEBOOLPARAMETER : BOOL
VAR_INPUT
	PINPUTDATA : POINTER TO BYTE;
	PARAMETER : DINT;
	PXVALUE : POINTER TO BOOL;
	XALLOWINVISIBLE : BOOL;
END_VAR
VAR_OUTPUT
	WERRORID : WORD;
END_VAR
END_METHOD

METHOD HLP_WRITEPARAMETER : BOOL
VAR_INPUT
	PINPUTDATA : POINTER TO BYTE;
	PARAMETER : DINT;
	PLRVALUE : POINTER TO LREAL;
	XALLOWINVISIBLE : BOOL;
END_VAR
VAR_OUTPUT
	WERRORID : WORD;
END_VAR
END_METHOD

METHOD HLP_INITPARREF : BOOL
VAR_INPUT
	PINPUTDATA : POINTER TO BYTE;
	PINPUTDATA2 : POINTER TO BYTE;
END_VAR
VAR_OUTPUT
	WERRORID : WORD;
END_VAR
END_METHOD

METHOD HLP_GETPARAMETERPROPERTIES : BOOL
VAR_INPUT
	PAXISREF : POINTER TO AXIS_REF;
	DIPARAMETER : DINT;
	XALLOWINVISIBLE : BOOL;
END_VAR
VAR_OUTPUT
	PPARAMADDR : POINTER TO BYTE := 0;
	EORDINALTYPE : L_MC1P_OrdinalType := L_MC1P_OrdinalType.otNONE;
	XREADWRITE : BOOL := FALSE;
	LRUNITFACTOR : LREAL := 0.0;
	LRDEFAULTVALUE : LREAL := 0.0;
	WVALUERANGES : WORD := 0;
	PVALUERANGES : POINTER TO L_MC1P_MinMaxValue := 0;
END_VAR
END_METHOD

(* ---- L_MC1P_PARAINTERFACE_AXIS_REF_ENC_UNIVERSAL.pou ---- *)
FUNCTION_BLOCK L_MC1P_PARAINTERFACE_AXIS_REF_ENC_UNIVERSAL
VAR
	ASCVALUERANGES : ARRAY [0..22] OF L_MC1P_MinMaxValue;
END_VAR
END_FUNCTION_BLOCK

METHOD HLP_READBOOLPARAMETER : BOOL
VAR_INPUT
	PINPUTDATA : POINTER TO BYTE;
	PARAMETER : DINT;
	PXVALUE : POINTER TO BOOL;
	XALLOWINVISIBLE : BOOL;
END_VAR
END_METHOD

METHOD HLP_READPARAMETER : BOOL
VAR_INPUT
	PINPUTDATA : POINTER TO BYTE;
	PARAMETER : DINT;
	PLRVALUE : POINTER TO LREAL;
	XALLOWINVISIBLE : BOOL;
END_VAR
END_METHOD

METHOD HLP_WRITEBOOLPARAMETER : BOOL
VAR_INPUT
	PINPUTDATA : POINTER TO BYTE;
	PARAMETER : DINT;
	PXVALUE : POINTER TO BOOL;
	XALLOWINVISIBLE : BOOL;
END_VAR
VAR_OUTPUT
	WERRORID : WORD;
END_VAR
END_METHOD

METHOD HLP_WRITEPARAMETER : BOOL
VAR_INPUT
	PINPUTDATA : POINTER TO BYTE;
	PARAMETER : DINT;
	PLRVALUE : POINTER TO LREAL;
	XALLOWINVISIBLE : BOOL;
END_VAR
VAR_OUTPUT
	WERRORID : WORD;
END_VAR
END_METHOD

METHOD HLP_INITPARREF : BOOL
VAR_INPUT
	PINPUTDATA : POINTER TO BYTE;
	PINPUTDATA2 : POINTER TO BYTE;
END_VAR
VAR_OUTPUT
	WERRORID : WORD;
END_VAR
END_METHOD

METHOD HLP_GETPARAMETERPROPERTIES : BOOL
VAR_INPUT
	PAXISREF : POINTER TO AXIS_REF;
	DIPARAMETER : DINT;
	XALLOWINVISIBLE : BOOL;
END_VAR
VAR_OUTPUT
	PPARAMADDR : POINTER TO BYTE := 0;
	EORDINALTYPE : L_MC1P_OrdinalType := L_MC1P_OrdinalType.otNONE;
	XREADWRITE : BOOL := FALSE;
	LRUNITFACTOR : LREAL := 0.0;
	LRDEFAULTVALUE : LREAL := 0.0;
	WVALUERANGES : WORD := 0;
	PVALUERANGES : POINTER TO L_MC1P_MinMaxValue := 0;
END_VAR
END_METHOD

(* ---- L_MC1P_PARAINTERFACE_AXIS_REF_GENERIC.pou ---- *)
FUNCTION_BLOCK L_MC1P_PARAINTERFACE_AXIS_REF_GENERIC
VAR
	ASCVALUERANGES : ARRAY [0..5] OF L_MC1P_MinMaxValue;
END_VAR
END_FUNCTION_BLOCK

METHOD HLP_READBOOLPARAMETER : BOOL
VAR_INPUT
	PINPUTDATA : POINTER TO BYTE;
	PARAMETER : DINT;
	PXVALUE : POINTER TO BOOL;
	XALLOWINVISIBLE : BOOL;
END_VAR
END_METHOD

METHOD HLP_READPARAMETER : BOOL
VAR_INPUT
	PINPUTDATA : POINTER TO BYTE;
	PARAMETER : DINT;
	PLRVALUE : POINTER TO LREAL;
	XALLOWINVISIBLE : BOOL;
END_VAR
END_METHOD

METHOD HLP_WRITEBOOLPARAMETER : BOOL
VAR_INPUT
	PINPUTDATA : POINTER TO BYTE;
	PARAMETER : DINT;
	PXVALUE : POINTER TO BOOL;
	XALLOWINVISIBLE : BOOL;
END_VAR
VAR_OUTPUT
	WERRORID : WORD;
END_VAR
END_METHOD

METHOD HLP_WRITEPARAMETER : BOOL
VAR_INPUT
	PINPUTDATA : POINTER TO BYTE;
	PARAMETER : DINT;
	PLRVALUE : POINTER TO LREAL;
	XALLOWINVISIBLE : BOOL;
END_VAR
VAR_OUTPUT
	WERRORID : WORD;
END_VAR
END_METHOD

METHOD HLP_INITPARREF : BOOL
VAR_INPUT
	PINPUTDATA : POINTER TO BYTE;
	PINPUTDATA2 : POINTER TO BYTE;
END_VAR
VAR_OUTPUT
	WERRORID : WORD;
END_VAR
END_METHOD

METHOD HLP_GETPARAMETERPROPERTIES : BOOL
VAR_INPUT
	PAXISREF : POINTER TO AXIS_REF;
	DIPARAMETER : DINT;
	XALLOWINVISIBLE : BOOL;
END_VAR
VAR_OUTPUT
	PPARAMADDR : POINTER TO BYTE := 0;
	EORDINALTYPE : L_MC1P_OrdinalType := L_MC1P_OrdinalType.otNONE;
	XREADWRITE : BOOL := FALSE;
	LRUNITFACTOR : LREAL := 0.0;
	LRDEFAULTVALUE : LREAL := 0.0;
	WVALUERANGES : WORD := 0;
	PVALUERANGES : POINTER TO L_MC1P_MinMaxValue := 0;
END_VAR
END_METHOD

(* ---- L_MC1P_PARAINTERFACE_AXIS_REF_I500_CAN.pou ---- *)
FUNCTION_BLOCK L_MC1P_PARAINTERFACE_AXIS_REF_I500_CAN
VAR
	ASCVALUERANGES : ARRAY [0..2] OF L_MC1P_MinMaxValue;
END_VAR
END_FUNCTION_BLOCK

METHOD HLP_READBOOLPARAMETER : BOOL
VAR_INPUT
	PINPUTDATA : POINTER TO BYTE;
	PARAMETER : DINT;
	PXVALUE : POINTER TO BOOL;
	XALLOWINVISIBLE : BOOL;
END_VAR
END_METHOD

METHOD HLP_READPARAMETER : BOOL
VAR_INPUT
	PINPUTDATA : POINTER TO BYTE;
	PARAMETER : DINT;
	PLRVALUE : POINTER TO LREAL;
	XALLOWINVISIBLE : BOOL;
END_VAR
END_METHOD

METHOD HLP_WRITEBOOLPARAMETER : BOOL
VAR_INPUT
	PINPUTDATA : POINTER TO BYTE;
	PARAMETER : DINT;
	PXVALUE : POINTER TO BOOL;
	XALLOWINVISIBLE : BOOL;
END_VAR
VAR_OUTPUT
	WERRORID : WORD;
END_VAR
END_METHOD

METHOD HLP_WRITEPARAMETER : BOOL
VAR_INPUT
	PINPUTDATA : POINTER TO BYTE;
	PARAMETER : DINT;
	PLRVALUE : POINTER TO LREAL;
	XALLOWINVISIBLE : BOOL;
END_VAR
VAR_OUTPUT
	WERRORID : WORD;
END_VAR
END_METHOD

METHOD HLP_INITPARREF : BOOL
VAR_INPUT
	PINPUTDATA : POINTER TO BYTE;
	PINPUTDATA2 : POINTER TO BYTE;
END_VAR
VAR_OUTPUT
	WERRORID : WORD;
END_VAR
END_METHOD

METHOD HLP_GETPARAMETERPROPERTIES : BOOL
VAR_INPUT
	PAXISREF : POINTER TO AXIS_REF;
	DIPARAMETER : DINT;
	XALLOWINVISIBLE : BOOL;
END_VAR
VAR_OUTPUT
	PPARAMADDR : POINTER TO BYTE := 0;
	EORDINALTYPE : L_MC1P_OrdinalType := L_MC1P_OrdinalType.otNONE;
	XREADWRITE : BOOL := FALSE;
	LRUNITFACTOR : LREAL := 0.0;
	LRDEFAULTVALUE : LREAL := 0.0;
	WVALUERANGES : WORD := 0;
	PVALUERANGES : POINTER TO L_MC1P_MinMaxValue := 0;
END_VAR
END_METHOD

(* ---- L_MC1P_PARAINTERFACE_AXIS_REF_I500_ETC.pou ---- *)
FUNCTION_BLOCK L_MC1P_PARAINTERFACE_AXIS_REF_I500_ETC
VAR
	ASCVALUERANGES : ARRAY [0..5] OF L_MC1P_MinMaxValue;
END_VAR
END_FUNCTION_BLOCK

METHOD HLP_READBOOLPARAMETER : BOOL
VAR_INPUT
	PINPUTDATA : POINTER TO BYTE;
	PARAMETER : DINT;
	PXVALUE : POINTER TO BOOL;
	XALLOWINVISIBLE : BOOL;
END_VAR
END_METHOD

METHOD HLP_READPARAMETER : BOOL
VAR_INPUT
	PINPUTDATA : POINTER TO BYTE;
	PARAMETER : DINT;
	PLRVALUE : POINTER TO LREAL;
	XALLOWINVISIBLE : BOOL;
END_VAR
END_METHOD

METHOD HLP_WRITEBOOLPARAMETER : BOOL
VAR_INPUT
	PINPUTDATA : POINTER TO BYTE;
	PARAMETER : DINT;
	PXVALUE : POINTER TO BOOL;
	XALLOWINVISIBLE : BOOL;
END_VAR
VAR_OUTPUT
	WERRORID : WORD;
END_VAR
END_METHOD

METHOD HLP_WRITEPARAMETER : BOOL
VAR_INPUT
	PINPUTDATA : POINTER TO BYTE;
	PARAMETER : DINT;
	PLRVALUE : POINTER TO LREAL;
	XALLOWINVISIBLE : BOOL;
END_VAR
VAR_OUTPUT
	WERRORID : WORD;
END_VAR
END_METHOD

METHOD HLP_INITPARREF : BOOL
VAR_INPUT
	PINPUTDATA : POINTER TO BYTE;
	PINPUTDATA2 : POINTER TO BYTE;
END_VAR
VAR_OUTPUT
	WERRORID : WORD;
END_VAR
END_METHOD

METHOD HLP_GETPARAMETERPROPERTIES : BOOL
VAR_INPUT
	PAXISREF : POINTER TO AXIS_REF;
	DIPARAMETER : DINT;
	XALLOWINVISIBLE : BOOL;
END_VAR
VAR_OUTPUT
	PPARAMADDR : POINTER TO BYTE := 0;
	EORDINALTYPE : L_MC1P_OrdinalType := L_MC1P_OrdinalType.otNONE;
	XREADWRITE : BOOL := FALSE;
	LRUNITFACTOR : LREAL := 0.0;
	LRDEFAULTVALUE : LREAL := 0.0;
	WVALUERANGES : WORD := 0;
	PVALUERANGES : POINTER TO L_MC1P_MinMaxValue := 0;
END_VAR
END_METHOD

(* ---- L_MC1P_PARAINTERFACE_AXIS_REF_I700.pou ---- *)
FUNCTION_BLOCK L_MC1P_PARAINTERFACE_AXIS_REF_I700
VAR
	ASCVALUERANGES : ARRAY [0..7] OF L_MC1P_MinMaxValue;
END_VAR
END_FUNCTION_BLOCK

METHOD HLP_READBOOLPARAMETER : BOOL
VAR_INPUT
	PINPUTDATA : POINTER TO BYTE;
	PARAMETER : DINT;
	PXVALUE : POINTER TO BOOL;
	XALLOWINVISIBLE : BOOL;
END_VAR
END_METHOD

METHOD HLP_READPARAMETER : BOOL
VAR_INPUT
	PINPUTDATA : POINTER TO BYTE;
	PARAMETER : DINT;
	PLRVALUE : POINTER TO LREAL;
	XALLOWINVISIBLE : BOOL;
END_VAR
END_METHOD

METHOD HLP_WRITEBOOLPARAMETER : BOOL
VAR_INPUT
	PINPUTDATA : POINTER TO BYTE;
	PARAMETER : DINT;
	PXVALUE : POINTER TO BOOL;
	XALLOWINVISIBLE : BOOL;
END_VAR
VAR_OUTPUT
	WERRORID : WORD;
END_VAR
END_METHOD

METHOD HLP_WRITEPARAMETER : BOOL
VAR_INPUT
	PINPUTDATA : POINTER TO BYTE;
	PARAMETER : DINT;
	PLRVALUE : POINTER TO LREAL;
	XALLOWINVISIBLE : BOOL;
END_VAR
VAR_OUTPUT
	WERRORID : WORD;
END_VAR
END_METHOD

METHOD HLP_INITPARREF : BOOL
VAR_INPUT
	PINPUTDATA : POINTER TO BYTE;
	PINPUTDATA2 : POINTER TO BYTE;
END_VAR
VAR_OUTPUT
	WERRORID : WORD;
END_VAR
END_METHOD

METHOD HLP_GETPARAMETERPROPERTIES : BOOL
VAR_INPUT
	PAXISREF : POINTER TO AXIS_REF;
	DIPARAMETER : DINT;
	XALLOWINVISIBLE : BOOL;
END_VAR
VAR_OUTPUT
	PPARAMADDR : POINTER TO BYTE := 0;
	EORDINALTYPE : L_MC1P_OrdinalType := L_MC1P_OrdinalType.otNONE;
	XREADWRITE : BOOL := FALSE;
	LRUNITFACTOR : LREAL := 0.0;
	LRDEFAULTVALUE : LREAL := 0.0;
	WVALUERANGES : WORD := 0;
	PVALUERANGES : POINTER TO L_MC1P_MinMaxValue := 0;
END_VAR
END_METHOD

(* ---- L_MC1P_PARAINTERFACE_AXIS_REF_I700_SLOT1.pou ---- *)
FUNCTION_BLOCK L_MC1P_PARAINTERFACE_AXIS_REF_I700_SLOT1
VAR
	ASCVALUERANGES : ARRAY [0..7] OF L_MC1P_MinMaxValue;
END_VAR
END_FUNCTION_BLOCK

METHOD HLP_READBOOLPARAMETER : BOOL
VAR_INPUT
	PINPUTDATA : POINTER TO BYTE;
	PARAMETER : DINT;
	PXVALUE : POINTER TO BOOL;
	XALLOWINVISIBLE : BOOL;
END_VAR
END_METHOD

METHOD HLP_READPARAMETER : BOOL
VAR_INPUT
	PINPUTDATA : POINTER TO BYTE;
	PARAMETER : DINT;
	PLRVALUE : POINTER TO LREAL;
	XALLOWINVISIBLE : BOOL;
END_VAR
END_METHOD

METHOD HLP_WRITEBOOLPARAMETER : BOOL
VAR_INPUT
	PINPUTDATA : POINTER TO BYTE;
	PARAMETER : DINT;
	PXVALUE : POINTER TO BOOL;
	XALLOWINVISIBLE : BOOL;
END_VAR
VAR_OUTPUT
	WERRORID : WORD;
END_VAR
END_METHOD

METHOD HLP_WRITEPARAMETER : BOOL
VAR_INPUT
	PINPUTDATA : POINTER TO BYTE;
	PARAMETER : DINT;
	PLRVALUE : POINTER TO LREAL;
	XALLOWINVISIBLE : BOOL;
END_VAR
VAR_OUTPUT
	WERRORID : WORD;
END_VAR
END_METHOD

METHOD HLP_INITPARREF : BOOL
VAR_INPUT
	PINPUTDATA : POINTER TO BYTE;
	PINPUTDATA2 : POINTER TO BYTE;
END_VAR
VAR_OUTPUT
	WERRORID : WORD;
END_VAR
END_METHOD

METHOD HLP_GETPARAMETERPROPERTIES : BOOL
VAR_INPUT
	PAXISREF : POINTER TO AXIS_REF;
	DIPARAMETER : DINT;
	XALLOWINVISIBLE : BOOL;
END_VAR
VAR_OUTPUT
	PPARAMADDR : POINTER TO BYTE := 0;
	EORDINALTYPE : L_MC1P_OrdinalType := L_MC1P_OrdinalType.otNONE;
	XREADWRITE : BOOL := FALSE;
	LRUNITFACTOR : LREAL := 0.0;
	LRDEFAULTVALUE : LREAL := 0.0;
	WVALUERANGES : WORD := 0;
	PVALUERANGES : POINTER TO L_MC1P_MinMaxValue := 0;
END_VAR
END_METHOD

(* ---- L_MC1P_PARAINTERFACE_AXIS_REF_I750.pou ---- *)
FUNCTION_BLOCK L_MC1P_PARAINTERFACE_AXIS_REF_I750
VAR
	ASCVALUERANGES : ARRAY [0..7] OF L_MC1P_MinMaxValue;
END_VAR
END_FUNCTION_BLOCK

METHOD HLP_READBOOLPARAMETER : BOOL
VAR_INPUT
	PINPUTDATA : POINTER TO BYTE;
	PARAMETER : DINT;
	PXVALUE : POINTER TO BOOL;
	XALLOWINVISIBLE : BOOL;
END_VAR
END_METHOD

METHOD HLP_READPARAMETER : BOOL
VAR_INPUT
	PINPUTDATA : POINTER TO BYTE;
	PARAMETER : DINT;
	PLRVALUE : POINTER TO LREAL;
	XALLOWINVISIBLE : BOOL;
END_VAR
END_METHOD

METHOD HLP_WRITEBOOLPARAMETER : BOOL
VAR_INPUT
	PINPUTDATA : POINTER TO BYTE;
	PARAMETER : DINT;
	PXVALUE : POINTER TO BOOL;
	XALLOWINVISIBLE : BOOL;
END_VAR
VAR_OUTPUT
	WERRORID : WORD;
END_VAR
END_METHOD

METHOD HLP_WRITEPARAMETER : BOOL
VAR_INPUT
	PINPUTDATA : POINTER TO BYTE;
	PARAMETER : DINT;
	PLRVALUE : POINTER TO LREAL;
	XALLOWINVISIBLE : BOOL;
END_VAR
VAR_OUTPUT
	WERRORID : WORD;
END_VAR
END_METHOD

METHOD HLP_INITPARREF : BOOL
VAR_INPUT
	PINPUTDATA : POINTER TO BYTE;
	PINPUTDATA2 : POINTER TO BYTE;
END_VAR
VAR_OUTPUT
	WERRORID : WORD;
END_VAR
END_METHOD

METHOD HLP_GETPARAMETERPROPERTIES : BOOL
VAR_INPUT
	PAXISREF : POINTER TO AXIS_REF;
	DIPARAMETER : DINT;
	XALLOWINVISIBLE : BOOL;
END_VAR
VAR_OUTPUT
	PPARAMADDR : POINTER TO BYTE := 0;
	EORDINALTYPE : L_MC1P_OrdinalType := L_MC1P_OrdinalType.otNONE;
	XREADWRITE : BOOL := FALSE;
	LRUNITFACTOR : LREAL := 0.0;
	LRDEFAULTVALUE : LREAL := 0.0;
	WVALUERANGES : WORD := 0;
	PVALUERANGES : POINTER TO L_MC1P_MinMaxValue := 0;
END_VAR
END_METHOD

(* ---- L_MC1P_PARAINTERFACE_AXIS_REF_I900.pou ---- *)
FUNCTION_BLOCK L_MC1P_PARAINTERFACE_AXIS_REF_I900
VAR
	ASCVALUERANGES : ARRAY [0..7] OF L_MC1P_MinMaxValue;
END_VAR
END_FUNCTION_BLOCK

METHOD HLP_READBOOLPARAMETER : BOOL
VAR_INPUT
	PINPUTDATA : POINTER TO BYTE;
	PARAMETER : DINT;
	PXVALUE : POINTER TO BOOL;
	XALLOWINVISIBLE : BOOL;
END_VAR
END_METHOD

METHOD HLP_READPARAMETER : BOOL
VAR_INPUT
	PINPUTDATA : POINTER TO BYTE;
	PARAMETER : DINT;
	PLRVALUE : POINTER TO LREAL;
	XALLOWINVISIBLE : BOOL;
END_VAR
END_METHOD

METHOD HLP_WRITEBOOLPARAMETER : BOOL
VAR_INPUT
	PINPUTDATA : POINTER TO BYTE;
	PARAMETER : DINT;
	PXVALUE : POINTER TO BOOL;
	XALLOWINVISIBLE : BOOL;
END_VAR
VAR_OUTPUT
	WERRORID : WORD;
END_VAR
END_METHOD

METHOD HLP_WRITEPARAMETER : BOOL
VAR_INPUT
	PINPUTDATA : POINTER TO BYTE;
	PARAMETER : DINT;
	PLRVALUE : POINTER TO LREAL;
	XALLOWINVISIBLE : BOOL;
END_VAR
VAR_OUTPUT
	WERRORID : WORD;
END_VAR
END_METHOD

METHOD HLP_INITPARREF : BOOL
VAR_INPUT
	PINPUTDATA : POINTER TO BYTE;
	PINPUTDATA2 : POINTER TO BYTE;
END_VAR
VAR_OUTPUT
	WERRORID : WORD;
END_VAR
END_METHOD

METHOD HLP_GETPARAMETERPROPERTIES : BOOL
VAR_INPUT
	PAXISREF : POINTER TO AXIS_REF;
	DIPARAMETER : DINT;
	XALLOWINVISIBLE : BOOL;
END_VAR
VAR_OUTPUT
	PPARAMADDR : POINTER TO BYTE := 0;
	EORDINALTYPE : L_MC1P_OrdinalType := L_MC1P_OrdinalType.otNONE;
	XREADWRITE : BOOL := FALSE;
	LRUNITFACTOR : LREAL := 0.0;
	LRDEFAULTVALUE : LREAL := 0.0;
	WVALUERANGES : WORD := 0;
	PVALUERANGES : POINTER TO L_MC1P_MinMaxValue := 0;
END_VAR
END_METHOD

(* ---- L_MC1P_PARAINTERFACE_AXIS_REF_I900_CIAADV.pou ---- *)
FUNCTION_BLOCK L_MC1P_PARAINTERFACE_AXIS_REF_I900_CIAADV
VAR
	ASCVALUERANGES : ARRAY [0..7] OF L_MC1P_MinMaxValue;
END_VAR
END_FUNCTION_BLOCK

METHOD HLP_READBOOLPARAMETER : BOOL
VAR_INPUT
	PINPUTDATA : POINTER TO BYTE;
	PARAMETER : DINT;
	PXVALUE : POINTER TO BOOL;
	XALLOWINVISIBLE : BOOL;
END_VAR
END_METHOD

METHOD HLP_READPARAMETER : BOOL
VAR_INPUT
	PINPUTDATA : POINTER TO BYTE;
	PARAMETER : DINT;
	PLRVALUE : POINTER TO LREAL;
	XALLOWINVISIBLE : BOOL;
END_VAR
END_METHOD

METHOD HLP_WRITEBOOLPARAMETER : BOOL
VAR_INPUT
	PINPUTDATA : POINTER TO BYTE;
	PARAMETER : DINT;
	PXVALUE : POINTER TO BOOL;
	XALLOWINVISIBLE : BOOL;
END_VAR
VAR_OUTPUT
	WERRORID : WORD;
END_VAR
END_METHOD

METHOD HLP_WRITEPARAMETER : BOOL
VAR_INPUT
	PINPUTDATA : POINTER TO BYTE;
	PARAMETER : DINT;
	PLRVALUE : POINTER TO LREAL;
	XALLOWINVISIBLE : BOOL;
END_VAR
VAR_OUTPUT
	WERRORID : WORD;
END_VAR
END_METHOD

METHOD HLP_INITPARREF : BOOL
VAR_INPUT
	PINPUTDATA : POINTER TO BYTE;
	PINPUTDATA2 : POINTER TO BYTE;
END_VAR
VAR_OUTPUT
	WERRORID : WORD;
END_VAR
END_METHOD

METHOD HLP_GETPARAMETERPROPERTIES : BOOL
VAR_INPUT
	PAXISREF : POINTER TO AXIS_REF;
	DIPARAMETER : DINT;
	XALLOWINVISIBLE : BOOL;
END_VAR
VAR_OUTPUT
	PPARAMADDR : POINTER TO BYTE := 0;
	EORDINALTYPE : L_MC1P_OrdinalType := L_MC1P_OrdinalType.otNONE;
	XREADWRITE : BOOL := FALSE;
	LRUNITFACTOR : LREAL := 0.0;
	LRDEFAULTVALUE : LREAL := 0.0;
	WVALUERANGES : WORD := 0;
	PVALUERANGES : POINTER TO L_MC1P_MinMaxValue := 0;
END_VAR
END_METHOD

(* ---- L_MC1P_PARAINTERFACE_AXIS_REF_I900_DRIVE.pou ---- *)
FUNCTION_BLOCK L_MC1P_PARAINTERFACE_AXIS_REF_I900_DRIVE
VAR
	ASCVALUERANGES : ARRAY [0..7] OF L_MC1P_MinMaxValue;
END_VAR
END_FUNCTION_BLOCK

METHOD HLP_READBOOLPARAMETER : BOOL
VAR_INPUT
	PINPUTDATA : POINTER TO BYTE;
	PARAMETER : DINT;
	PXVALUE : POINTER TO BOOL;
	XALLOWINVISIBLE : BOOL;
END_VAR
END_METHOD

METHOD HLP_READPARAMETER : BOOL
VAR_INPUT
	PINPUTDATA : POINTER TO BYTE;
	PARAMETER : DINT;
	PLRVALUE : POINTER TO LREAL;
	XALLOWINVISIBLE : BOOL;
END_VAR
END_METHOD

METHOD HLP_WRITEBOOLPARAMETER : BOOL
VAR_INPUT
	PINPUTDATA : POINTER TO BYTE;
	PARAMETER : DINT;
	PXVALUE : POINTER TO BOOL;
	XALLOWINVISIBLE : BOOL;
END_VAR
VAR_OUTPUT
	WERRORID : WORD;
END_VAR
END_METHOD

METHOD HLP_WRITEPARAMETER : BOOL
VAR_INPUT
	PINPUTDATA : POINTER TO BYTE;
	PARAMETER : DINT;
	PLRVALUE : POINTER TO LREAL;
	XALLOWINVISIBLE : BOOL;
END_VAR
VAR_OUTPUT
	WERRORID : WORD;
END_VAR
END_METHOD

METHOD HLP_INITPARREF : BOOL
VAR_INPUT
	PINPUTDATA : POINTER TO BYTE;
	PINPUTDATA2 : POINTER TO BYTE;
END_VAR
VAR_OUTPUT
	WERRORID : WORD;
END_VAR
END_METHOD

METHOD HLP_GETPARAMETERPROPERTIES : BOOL
VAR_INPUT
	PAXISREF : POINTER TO AXIS_REF;
	DIPARAMETER : DINT;
	XALLOWINVISIBLE : BOOL;
END_VAR
VAR_OUTPUT
	PPARAMADDR : POINTER TO BYTE := 0;
	EORDINALTYPE : L_MC1P_OrdinalType := L_MC1P_OrdinalType.otNONE;
	XREADWRITE : BOOL := FALSE;
	LRUNITFACTOR : LREAL := 0.0;
	LRDEFAULTVALUE : LREAL := 0.0;
	WVALUERANGES : WORD := 0;
	PVALUERANGES : POINTER TO L_MC1P_MinMaxValue := 0;
END_VAR
END_METHOD

(* ---- L_MC1P_PARAINTERFACE_AXIS_REF_I900_DRIVE_CIA.pou ---- *)
FUNCTION_BLOCK L_MC1P_PARAINTERFACE_AXIS_REF_I900_DRIVE_CIA
VAR
	ASCVALUERANGES : ARRAY [0..7] OF L_MC1P_MinMaxValue;
END_VAR
END_FUNCTION_BLOCK

METHOD HLP_READBOOLPARAMETER : BOOL
VAR_INPUT
	PINPUTDATA : POINTER TO BYTE;
	PARAMETER : DINT;
	PXVALUE : POINTER TO BOOL;
	XALLOWINVISIBLE : BOOL;
END_VAR
END_METHOD

METHOD HLP_READPARAMETER : BOOL
VAR_INPUT
	PINPUTDATA : POINTER TO BYTE;
	PARAMETER : DINT;
	PLRVALUE : POINTER TO LREAL;
	XALLOWINVISIBLE : BOOL;
END_VAR
END_METHOD

METHOD HLP_WRITEBOOLPARAMETER : BOOL
VAR_INPUT
	PINPUTDATA : POINTER TO BYTE;
	PARAMETER : DINT;
	PXVALUE : POINTER TO BOOL;
	XALLOWINVISIBLE : BOOL;
END_VAR
VAR_OUTPUT
	WERRORID : WORD;
END_VAR
END_METHOD

METHOD HLP_WRITEPARAMETER : BOOL
VAR_INPUT
	PINPUTDATA : POINTER TO BYTE;
	PARAMETER : DINT;
	PLRVALUE : POINTER TO LREAL;
	XALLOWINVISIBLE : BOOL;
END_VAR
VAR_OUTPUT
	WERRORID : WORD;
END_VAR
END_METHOD

METHOD HLP_INITPARREF : BOOL
VAR_INPUT
	PINPUTDATA : POINTER TO BYTE;
	PINPUTDATA2 : POINTER TO BYTE;
END_VAR
VAR_OUTPUT
	WERRORID : WORD;
END_VAR
END_METHOD

METHOD HLP_GETPARAMETERPROPERTIES : BOOL
VAR_INPUT
	PAXISREF : POINTER TO AXIS_REF;
	DIPARAMETER : DINT;
	XALLOWINVISIBLE : BOOL;
END_VAR
VAR_OUTPUT
	PPARAMADDR : POINTER TO BYTE := 0;
	EORDINALTYPE : L_MC1P_OrdinalType := L_MC1P_OrdinalType.otNONE;
	XREADWRITE : BOOL := FALSE;
	LRUNITFACTOR : LREAL := 0.0;
	LRDEFAULTVALUE : LREAL := 0.0;
	WVALUERANGES : WORD := 0;
	PVALUERANGES : POINTER TO L_MC1P_MinMaxValue := 0;
END_VAR
END_METHOD

(* ---- L_MC1P_PARAINTERFACE_AXIS_REF_UNIVERSAL.pou ---- *)
FUNCTION_BLOCK L_MC1P_PARAINTERFACE_AXIS_REF_UNIVERSAL
VAR
	ASCVALUERANGES : ARRAY [0..7] OF L_MC1P_MinMaxValue;
END_VAR
END_FUNCTION_BLOCK

METHOD HLP_READBOOLPARAMETER : BOOL
VAR_INPUT
	PINPUTDATA : POINTER TO BYTE;
	PARAMETER : DINT;
	PXVALUE : POINTER TO BOOL;
	XALLOWINVISIBLE : BOOL;
END_VAR
END_METHOD

METHOD HLP_READPARAMETER : BOOL
VAR_INPUT
	PINPUTDATA : POINTER TO BYTE;
	PARAMETER : DINT;
	PLRVALUE : POINTER TO LREAL;
	XALLOWINVISIBLE : BOOL;
END_VAR
END_METHOD

METHOD HLP_WRITEBOOLPARAMETER : BOOL
VAR_INPUT
	PINPUTDATA : POINTER TO BYTE;
	PARAMETER : DINT;
	PXVALUE : POINTER TO BOOL;
	XALLOWINVISIBLE : BOOL;
END_VAR
VAR_OUTPUT
	WERRORID : WORD;
END_VAR
END_METHOD

METHOD HLP_WRITEPARAMETER : BOOL
VAR_INPUT
	PINPUTDATA : POINTER TO BYTE;
	PARAMETER : DINT;
	PLRVALUE : POINTER TO LREAL;
	XALLOWINVISIBLE : BOOL;
END_VAR
VAR_OUTPUT
	WERRORID : WORD;
END_VAR
END_METHOD

METHOD HLP_INITPARREF : BOOL
VAR_INPUT
	PINPUTDATA : POINTER TO BYTE;
	PINPUTDATA2 : POINTER TO BYTE;
END_VAR
VAR_OUTPUT
	WERRORID : WORD;
END_VAR
END_METHOD

METHOD HLP_GETPARAMETERPROPERTIES : BOOL
VAR_INPUT
	PAXISREF : POINTER TO AXIS_REF;
	DIPARAMETER : DINT;
	XALLOWINVISIBLE : BOOL;
END_VAR
VAR_OUTPUT
	PPARAMADDR : POINTER TO BYTE := 0;
	EORDINALTYPE : L_MC1P_OrdinalType := L_MC1P_OrdinalType.otNONE;
	XREADWRITE : BOOL := FALSE;
	LRUNITFACTOR : LREAL := 0.0;
	LRDEFAULTVALUE : LREAL := 0.0;
	WVALUERANGES : WORD := 0;
	PVALUERANGES : POINTER TO L_MC1P_MinMaxValue := 0;
END_VAR
END_METHOD

(* ---- L_MC1P_PARAINTERFACE_AXIS_REF_VIRTUAL.pou ---- *)
FUNCTION_BLOCK L_MC1P_PARAINTERFACE_AXIS_REF_VIRTUAL
VAR
	ASCVALUERANGES : ARRAY [0..5] OF L_MC1P_MinMaxValue;
END_VAR
END_FUNCTION_BLOCK

METHOD HLP_READBOOLPARAMETER : BOOL
VAR_INPUT
	PINPUTDATA : POINTER TO BYTE;
	PARAMETER : DINT;
	PXVALUE : POINTER TO BOOL;
	XALLOWINVISIBLE : BOOL;
END_VAR
END_METHOD

METHOD HLP_READPARAMETER : BOOL
VAR_INPUT
	PINPUTDATA : POINTER TO BYTE;
	PARAMETER : DINT;
	PLRVALUE : POINTER TO LREAL;
	XALLOWINVISIBLE : BOOL;
END_VAR
END_METHOD

METHOD HLP_WRITEBOOLPARAMETER : BOOL
VAR_INPUT
	PINPUTDATA : POINTER TO BYTE;
	PARAMETER : DINT;
	PXVALUE : POINTER TO BOOL;
	XALLOWINVISIBLE : BOOL;
END_VAR
VAR_OUTPUT
	WERRORID : WORD;
END_VAR
END_METHOD

METHOD HLP_WRITEPARAMETER : BOOL
VAR_INPUT
	PINPUTDATA : POINTER TO BYTE;
	PARAMETER : DINT;
	PLRVALUE : POINTER TO LREAL;
	XALLOWINVISIBLE : BOOL;
END_VAR
VAR_OUTPUT
	WERRORID : WORD;
END_VAR
END_METHOD

METHOD HLP_INITPARREF : BOOL
VAR_INPUT
	PINPUTDATA : POINTER TO BYTE;
	PINPUTDATA2 : POINTER TO BYTE;
END_VAR
VAR_OUTPUT
	WERRORID : WORD;
END_VAR
END_METHOD

METHOD HLP_GETPARAMETERPROPERTIES : BOOL
VAR_INPUT
	PAXISREF : POINTER TO AXIS_REF;
	DIPARAMETER : DINT;
	XALLOWINVISIBLE : BOOL;
END_VAR
VAR_OUTPUT
	PPARAMADDR : POINTER TO BYTE := 0;
	EORDINALTYPE : L_MC1P_OrdinalType := L_MC1P_OrdinalType.otNONE;
	XREADWRITE : BOOL := FALSE;
	LRUNITFACTOR : LREAL := 0.0;
	LRDEFAULTVALUE : LREAL := 0.0;
	WVALUERANGES : WORD := 0;
	PVALUERANGES : POINTER TO L_MC1P_MinMaxValue := 0;
END_VAR
END_METHOD

(* ---- L_MC1P_PARAINTERFACE_AXIS_REF_VIRTUALM_I900.pou ---- *)
FUNCTION_BLOCK L_MC1P_PARAINTERFACE_AXIS_REF_VIRTUALM_I900
VAR
	ASCVALUERANGES : ARRAY [0..3] OF L_MC1P_MinMaxValue;
END_VAR
END_FUNCTION_BLOCK

METHOD HLP_READBOOLPARAMETER : BOOL
VAR_INPUT
	PINPUTDATA : POINTER TO BYTE;
	PARAMETER : DINT;
	PXVALUE : POINTER TO BOOL;
	XALLOWINVISIBLE : BOOL;
END_VAR
END_METHOD

METHOD HLP_READPARAMETER : BOOL
VAR_INPUT
	PINPUTDATA : POINTER TO BYTE;
	PARAMETER : DINT;
	PLRVALUE : POINTER TO LREAL;
	XALLOWINVISIBLE : BOOL;
END_VAR
END_METHOD

METHOD HLP_WRITEBOOLPARAMETER : BOOL
VAR_INPUT
	PINPUTDATA : POINTER TO BYTE;
	PARAMETER : DINT;
	PXVALUE : POINTER TO BOOL;
	XALLOWINVISIBLE : BOOL;
END_VAR
VAR_OUTPUT
	WERRORID : WORD;
END_VAR
END_METHOD

METHOD HLP_WRITEPARAMETER : BOOL
VAR_INPUT
	PINPUTDATA : POINTER TO BYTE;
	PARAMETER : DINT;
	PLRVALUE : POINTER TO LREAL;
	XALLOWINVISIBLE : BOOL;
END_VAR
VAR_OUTPUT
	WERRORID : WORD;
END_VAR
END_METHOD

METHOD HLP_INITPARREF : BOOL
VAR_INPUT
	PINPUTDATA : POINTER TO BYTE;
	PINPUTDATA2 : POINTER TO BYTE;
END_VAR
VAR_OUTPUT
	WERRORID : WORD;
END_VAR
END_METHOD

METHOD HLP_GETPARAMETERPROPERTIES : BOOL
VAR_INPUT
	PAXISREF : POINTER TO AXIS_REF;
	DIPARAMETER : DINT;
	XALLOWINVISIBLE : BOOL;
END_VAR
VAR_OUTPUT
	PPARAMADDR : POINTER TO BYTE := 0;
	EORDINALTYPE : L_MC1P_OrdinalType := L_MC1P_OrdinalType.otNONE;
	XREADWRITE : BOOL := FALSE;
	LRUNITFACTOR : LREAL := 0.0;
	LRDEFAULTVALUE : LREAL := 0.0;
	WVALUERANGES : WORD := 0;
	PVALUERANGES : POINTER TO L_MC1P_MinMaxValue := 0;
END_VAR
END_METHOD

(* ---- L_MC1P_PARAINTERFACE_AXIS_REF_VMA.pou ---- *)
FUNCTION_BLOCK L_MC1P_PARAINTERFACE_AXIS_REF_VMA
VAR
	ASCVALUERANGES : ARRAY [0..5] OF L_MC1P_MinMaxValue;
END_VAR
END_FUNCTION_BLOCK

METHOD HLP_READBOOLPARAMETER : BOOL
VAR_INPUT
	PINPUTDATA : POINTER TO BYTE;
	PARAMETER : DINT;
	PXVALUE : POINTER TO BOOL;
	XALLOWINVISIBLE : BOOL;
END_VAR
END_METHOD

METHOD HLP_READPARAMETER : BOOL
VAR_INPUT
	PINPUTDATA : POINTER TO BYTE;
	PARAMETER : DINT;
	PLRVALUE : POINTER TO LREAL;
	XALLOWINVISIBLE : BOOL;
END_VAR
END_METHOD

METHOD HLP_WRITEBOOLPARAMETER : BOOL
VAR_INPUT
	PINPUTDATA : POINTER TO BYTE;
	PARAMETER : DINT;
	PXVALUE : POINTER TO BOOL;
	XALLOWINVISIBLE : BOOL;
END_VAR
VAR_OUTPUT
	WERRORID : WORD;
END_VAR
END_METHOD

METHOD HLP_WRITEPARAMETER : BOOL
VAR_INPUT
	PINPUTDATA : POINTER TO BYTE;
	PARAMETER : DINT;
	PLRVALUE : POINTER TO LREAL;
	XALLOWINVISIBLE : BOOL;
END_VAR
VAR_OUTPUT
	WERRORID : WORD;
END_VAR
END_METHOD

METHOD HLP_INITPARREF : BOOL
VAR_INPUT
	PINPUTDATA : POINTER TO BYTE;
	PINPUTDATA2 : POINTER TO BYTE;
END_VAR
VAR_OUTPUT
	WERRORID : WORD;
END_VAR
END_METHOD

METHOD HLP_GETPARAMETERPROPERTIES : BOOL
VAR_INPUT
	PAXISREF : POINTER TO AXIS_REF;
	DIPARAMETER : DINT;
	XALLOWINVISIBLE : BOOL;
END_VAR
VAR_OUTPUT
	PPARAMADDR : POINTER TO BYTE := 0;
	EORDINALTYPE : L_MC1P_OrdinalType := L_MC1P_OrdinalType.otNONE;
	XREADWRITE : BOOL := FALSE;
	LRUNITFACTOR : LREAL := 0.0;
	LRDEFAULTVALUE : LREAL := 0.0;
	WVALUERANGES : WORD := 0;
	PVALUERANGES : POINTER TO L_MC1P_MinMaxValue := 0;
END_VAR
END_METHOD

(* ---- L_MC1P_PARSIM.pou ---- *)
FUNCTION_BLOCK L_MC1P_PARSIM
VAR
	C_ERROR_NOERROR : WORD := 0;
	C_ERROR_NOPARAMETERDATABASE : WORD := 1;
	C_ERROR_DATATYPENOTSUPPORTED : WORD := 2;
	C_ERROR_PARAMETERDOESNOTEXIST : WORD := 3;
	C_ERROR_INVALIDINUTDATA : WORD := 4;
	C_ERROR_BUFFERTOSMALL : WORD := 5;
	C_ERROR_NOWRITEACCESS : WORD := 6;
	C_ERROR_SIZEMISMATCH : WORD := 7;
END_VAR
END_FUNCTION_BLOCK

(* ---- L_MC1P_PARSIMREAD.pou ---- *)
FUNCTION_BLOCK L_MC1P_PARSIMREAD EXTENDS L_MC1P_ParSim
VAR_INPUT
	XEXECUTE : BOOL;
	WINDEX : WORD;
	BYSUBINDEX : BYTE;
	PBUFFER : POINTER TO BYTE;
	SZSIZE : CAA_SIZE;
	UDITIMEOUT : UDINT;
	PPARAMDATA : POINTER TO L_MC1P_ParameterDataSim;
	WPARAMCOUNT : WORD;
	XSLOTB : BOOL;
	LRDELAY : LREAL := 0.01;
	LRTASKCYCLE : LREAL;
END_VAR
VAR_OUTPUT
	XBUSY : BOOL;
	XDONE : BOOL;
	XERROR : BOOL;
	EERRORCODE : WORD;
	SZDATAREAD : CAA_SIZE;
END_VAR
VAR
	XEXECUTEOLD : BOOL;
	XRESETOUTPUT : BOOL;
	IDX : WORD;
	XFOUND : BOOL;
	LRWAITCOUNTER : LREAL;
	WSEARCHINDEX : WORD := 0;
END_VAR
END_FUNCTION_BLOCK

METHOD GETVALUE : L_UBUP_VarValue
VAR_INPUT
	PSRCVALUE : POINTER TO L_UBUP_VarValue;
	PDESTVALUE : POINTER TO L_UBUP_VarValue;
	EFIXTOLREAL : L_MC1P_ScaleFixToLREAL;
	BYNROFBYTE : BYTE;
END_VAR
VAR_OUTPUT
	EERRORCODE : WORD;
	SZDATAREAD : CAA_SIZE;
END_VAR
END_METHOD

(* ---- L_MC1P_PARSIMWRITE.pou ---- *)
FUNCTION_BLOCK L_MC1P_PARSIMWRITE EXTENDS L_MC1P_ParSim
VAR_INPUT
	XEXECUTE : BOOL;
	WINDEX : WORD;
	BYSUBINDEX : BYTE;
	PBUFFER : POINTER TO BYTE;
	SZSIZE : CAA_SIZE;
	UDITIMEOUT : UDINT;
	PPARAMDATA : POINTER TO L_MC1P_ParameterDataSim;
	WPARAMCOUNT : WORD;
	XSLOTB : BOOL;
	LRDELAY : LREAL := 0.01;
	LRTASKCYCLE : LREAL;
END_VAR
VAR_OUTPUT
	XBUSY : BOOL;
	XDONE : BOOL;
	XERROR : BOOL;
	EERRORCODE : WORD;
END_VAR
VAR
	XEXECUTEOLD : BOOL;
	XRESETOUTPUT : BOOL;
	IDX : WORD;
	XFOUND : BOOL;
	LRWAITCOUNTER : LREAL;
	PTEMPVALUE : POINTER TO L_UBUP_VarValue;
	TEMPVALUEDEST : L_UBUP_VarValue;
	WSEARCHINDEX : WORD := 0;
END_VAR
END_FUNCTION_BLOCK

METHOD SETVALUE : L_UBUP_VarValue
VAR_INPUT
	PSRCVALUE : POINTER TO L_UBUP_VarValue;
	PDESTVALUE : POINTER TO L_UBUP_VarValue;
	EFIXTOLREAL : L_MC1P_ScaleFixToLREAL;
	BYNROFBYTE : BYTE;
END_VAR
VAR_OUTPUT
	EERRORCODE : WORD;
END_VAR
END_METHOD

(* ---- L_MC1P_POLEPOSITIONIDENTIFICATION.pou ---- *)
FUNCTION_BLOCK L_MC1P_POLEPOSITIONIDENTIFICATION EXTENDS L_MC1P_Template
VAR_INPUT
	XENABLE : BOOL;
	XEXECUTEPPI : BOOL := FALSE;
	XABORTPPI : BOOL := FALSE;
	XSETPOLEPOSITION : BOOL := FALSE;
	XRESETPOLEPOSITION : BOOL := FALSE;
END_VAR
VAR_OUTPUT
	XDONE : BOOL := FALSE;
	XBUSY : BOOL := FALSE;
	XACTIVE : BOOL := FALSE;
	XCOMMANDABORTED : BOOL := FALSE;
	XERROR : BOOL := FALSE;
	EERRORID : L_IE1P_Error;
	XPPINVALID : BOOL := FALSE;
END_VAR
VAR
	WFUNID : WORD;
	XENABLEOLD : BOOL;
	XRESETOUTPUT : BOOL;
	PAXISREAL : POINTER TO _AXIS_REF_REAL;
	MC_WRITEPARAMETER1 : MC_writeParameter;
	LROPERATIONMODE : LREAL;
	XREGULATORON : BOOL := FALSE;
	XPOWSTATUS : BOOL := FALSE;
	XPOWVALID : BOOL := FALSE;
	XSETPOLEPOSITIONOLD : BOOL := FALSE;
	XRESETPOLEPOSITIONOLD : BOOL := FALSE;
	XEXECUTEPPIOLD : BOOL := FALSE;
	WFBID : WORD := 0;
	ITFPLIACCESS : L_MC1P_IPLIAccess;
	WPPISTATE : WORD := 0;
	WPPIMODE : WORD := 0;
	TON : ton;
	XDISABLING : BOOL := FALSE;
	XOPERATIONMODESWITCHED : BOOL := FALSE;
	POWERRORID : L_IE1P_Error := L_IE1P_Error.NoError;
	BYDRIVESTATEOLD : BYTE;
	XSETREGULATORONFALSE : BOOL := FALSE;
	XABORTPPIOLD : BOOL := FALSE;
	XABORTING : BOOL := FALSE;
END_VAR
END_FUNCTION_BLOCK

(* ---- L_MC1P_POSCONTROLEXTENCODER.pou ---- *)
FUNCTION_BLOCK L_MC1P_POSCONTROLEXTENCODER EXTENDS L_MC1P_Template
VAR_INPUT
	XENABLE : BOOL;
	ENCODERAXIS : L_MC1P_IEncoderInterface;
	XACTIVATEENCODER : BOOL;
	LRGAIN : LREAL := 20.0;
	LROUTPUTLIMITATION : LREAL := 10000.0;
END_VAR
VAR_OUTPUT
	XBUSY : BOOL;
	XERROR : BOOL;
	EERRORID : L_IE1P_Error;
	EACTIVECONTROLMODE : L_MC1P_ControlMode := L_MC1P_ControlMode.PosCtrlDrive;
END_VAR
VAR
	XENABLEOLD : BOOL;
	PXDUMMY : POINTER TO BOOL;
	ENCODERAXISOLD : L_MC1P_IEncoderInterface;
	PSDUMMY : POINTER TO STRING;
	PAXIS : POINTER TO _AXIS_REF_REAL;
	PAXISENC : POINTER TO _AXIS_REF_REAL;
	XACTIVATEEXTENCODEROLD : BOOL;
	LRACTPOSENC : LREAL;
	LRACTENCROUNDS : LREAL;
	XTMP : BOOL;
	PLRDUMMY : POINTER TO LREAL;
END_VAR
END_FUNCTION_BLOCK

(* ---- L_MC1P_POSCONTROLLER.pou ---- *)
FUNCTION_BLOCK L_MC1P_POSCONTROLLER
VAR_INPUT
	LRGAIN : LREAL;
	LROUTPUTLIMITATION : LREAL;
	LRADAPT : LREAL := 1;
	LRADAPTINTERNAL : LREAL := 1;
END_VAR
VAR_OUTPUT
	LROUTPUT : LREAL;
END_VAR
VAR
	LRDELTAPOSOUT : LREAL;
	LRPOSCTRLOUTLIMIT : LREAL := 3600;
	LRVPPOSCTRL : LREAL;
	XLIMITED : BOOL;
	POSCONTROLLERLIMITED : BOOL;
END_VAR
END_FUNCTION_BLOCK

METHOD CALCCONTROLLER
VAR_INPUT
	LRSETPOSITION : LREAL;
	LRSETVELOCITY : LREAL;
	LRSETACCELERATION : LREAL;
	LRSETTORQUE : LREAL;
	LRSETJERK : LREAL;
	LRACTPOSITIONIN : LREAL;
	LRACTVELOCITYIN : LREAL;
	LRACTACCELERATIONIN : LREAL;
	LRACTTORQUEIN : LREAL;
END_VAR
VAR_OUTPUT
	LRSETPOSITIONOUT : LREAL;
	LRSETVELOCITYOUT : LREAL;
	LRSETACCELERATIONOUT : LREAL;
	LRSETTORQUEOUT : LREAL;
END_VAR
VAR_IN_OUT
	AXIS : _AXIS_REF_REAL;
END_VAR
END_METHOD

METHOD POSCONTROL : LREAL
VAR_INPUT
	LRDELTAPOS : LREAL;
END_VAR
VAR_OUTPUT
	XLIMIT : BOOL;
END_VAR
VAR_IN_OUT
	AXIS : _AXIS_REF_REAL;
END_VAR
END_METHOD

(* ---- L_MC1P_POSCONTROLLERV2.pou ---- *)
FUNCTION_BLOCK L_MC1P_POSCONTROLLERV2
VAR_INPUT
	LRGAIN : LREAL := 20;
	LROUTPUTLIMITATION : LREAL := 600000;
	LRADAPT : LREAL := 1;
	LRADAPTINTERNAL : LREAL := 1;
	XENABLEDELAYFACTOR : BOOL := TRUE;
	LRADDDELAYFACTOR : LREAL := 0;
	XDISABLEPOSCTRLINPUTLIMITATION : BOOL;
	ITFPOSCTRLADAPTCURVE : L_MC1P_IControllerAdaption;
END_VAR
VAR_OUTPUT
	LROUTPUT : LREAL;
	LRDELTAPOSOUT : LREAL;
	LRADAPTACTIVE : LREAL;
END_VAR
VAR
	DWTIMEDIFF : DWORD;
	LRDELAYFACTOR : LREAL;
	LRPOSCTRLOUTLIMIT : LREAL := 3600;
	LRVPPOSCTRL : LREAL;
	LRDELAYFACTORINT : LREAL;
	ALRSETPOS : ARRAY [0..15] OF LREAL;
	ALRSETPOSROUNDS : ARRAY [0..15] OF LREAL;
	IDX : WORD;
	XINIT : BOOL := TRUE;
	XBUFFER : BOOL;
	LRSETPOSITIONTMP : LREAL;
	LRSETROUNDSTMP : LREAL;
	LRCOMPMODROUNDS : LREAL;
	LRFACTOR : LREAL;
	WUPPERIDX : WORD;
	WLOWERIDX : WORD;
	LRDELTAROUNDSTMP : LREAL;
	LRDELTAPOSTMP : LREAL;
	DWLASTCALLTIME : DWORD;
	XLIMITED : BOOL;
	LRINITIALPOSDELTA : LREAL;
	XINPUTLIMITATIONACTIVE : BOOL;
	POSCONTROLLERLIMITED : BOOL;
END_VAR
END_FUNCTION_BLOCK

METHOD CALCCONTROLLER
VAR_INPUT
	LRSETPOSITION : LREAL;
	LRSETVELOCITY : LREAL;
	LRSETACCELERATION : LREAL;
	LRSETTORQUE : LREAL;
	LRSETJERK : LREAL;
	LRACTPOSITIONIN : LREAL;
	LRACTVELOCITYIN : LREAL;
	LRACTACCELERATIONIN : LREAL;
	LRACTTORQUEIN : LREAL;
END_VAR
VAR_OUTPUT
	LRSETPOSITIONOUT : LREAL;
	LRSETVELOCITYOUT : LREAL;
	LRSETACCELERATIONOUT : LREAL;
	LRSETTORQUEOUT : LREAL;
END_VAR
VAR_IN_OUT
	AXIS : _AXIS_REF_REAL;
END_VAR
END_METHOD

METHOD POSCONTROL : LREAL
VAR_INPUT
	LRDELTAPOS : LREAL;
END_VAR
VAR_OUTPUT
	XLIMIT : BOOL;
END_VAR
VAR_IN_OUT
	AXIS : _AXIS_REF_REAL;
END_VAR
END_METHOD

(* ---- L_MC1P_POSCTRLADAPTIONCURVE.pou ---- *)
FUNCTION_BLOCK L_MC1P_POSCTRLADAPTIONCURVE
VAR_INPUT
	XACTIVATEGAINADAPTIONCURVE : BOOL := FALSE;
	XDATAPOINTSVALID : BOOL := TRUE;
	AWPARPOSGAINADAPTSPEED : ARRAY [1..5] OF WORD := [10, 100, 1000, 2000, 5000];
	AWPARPOSGAINADAPTOUT : ARRAY [1..5] OF WORD := [100, 100, 100, 100, 100];
END_VAR
END_FUNCTION_BLOCK

METHOD CALCADAPTIONCURVE : LREAL
VAR_INPUT
	LRSETVEL : LREAL;
END_VAR
VAR_IN_OUT
	AXIS : _AXIS_REF_REAL;
END_VAR
END_METHOD

METHOD CALCULATEPOINT : LREAL
VAR_IN_OUT
	WXACT : WORD;
	WXSTART : WORD;
	WXEND : WORD;
	WYSTART : WORD;
	WYEND : WORD;
END_VAR
END_METHOD

(* ---- L_MC1P_POSGENERATOR.pou ---- *)
FUNCTION_BLOCK L_MC1P_POSGENERATOR
VAR_INPUT
	XENABLE : BOOL;
	XEXECUTE : BOOL;
	XABORTPROFILE : BOOL;
	LRCORRECTION : LREAL;
	LRMAXVELPOS : LREAL := 10;
	LRMAXVELNEG : LREAL := 10;
	LRACCDEC : LREAL := 100;
	EPROFILETYPE : L_MC1P_ProfileType := 0;
END_VAR
VAR_OUTPUT
	LRPOSOUTUNLIMITED : LREAL;
	LRRESIDUALOFFSET : LREAL;
	LRSPEEDOUT : LREAL;
	XPROFILEFAILED : BOOL;
	XPROFILEABORTED : BOOL;
	XINTARGET : BOOL;
	XBUSY : BOOL;
	DISTATE : DINT;
END_VAR
VAR_IN_OUT
	AXIS : Axis_REF;
END_VAR
VAR
	L_SDINTEGRATE1 : L_USPP_Integrate;
	R_TRIG1 : R_TRIG;
	R_TRIG2 : R_TRIG;
	F_TRIG2 : F_TRIG;
	F_TRIG3 : F_TRIG;
	DWPOSMODE : DWORD := 1;
	DWDISABLEMODE : DWORD;
	LRRAMPDISTANCE : LREAL;
	LRDELTAY : LREAL;
	LRBASICPOSITION : LREAL;
	BYSTEP : BYTE;
	BNEGSPEEDSELECTED : BOOL;
	LRXNORM : LREAL;
	LRPOSOUTOLD : LREAL;
	N : INT;
	LRMAXSPEEDINTERN : LREAL;
	LRMAXSPEEDNEG : LREAL;
	LRMAXSPEEDPOS : LREAL;
	LRSTARTPOSITION : LREAL;
	XSAVESTARTPOSITION : BOOL;
	LRPOSOUT : LREAL;
	LRPOSOUTOLDTEST : LREAL;
	LRPOSTEST : LREAL;
	XENDOFPROFILE : BOOL;
END_VAR
END_FUNCTION_BLOCK

METHOD A01_PROFILECONTROL
END_METHOD

METHOD A02_POLYNOMIAL4THORDER
END_METHOD

METHOD A03_POLYNOMIAL2NDORDER
END_METHOD

METHOD A04_POLYNOMIAL5THORDER
END_METHOD

(* ---- L_MC1P_POSGENERATORABORTCORRECTION.pou ---- *)
FUNCTION_BLOCK L_MC1P_POSGENERATORABORTCORRECTION
VAR_INPUT
	XENABLE : BOOL;
	LRCYCLETIME : LREAL;
	XABORTFROMPOSCTRL : BOOL;
	LRMAXACC : LREAL;
	LRACTVELFROMPOSCTRL : LREAL;
	LRSIMPLEPOSUNLIMITED : LREAL;
END_VAR
VAR_OUTPUT
	XABORTPROFILEFINISHED : BOOL;
	LRPOSOUT : LREAL;
END_VAR
VAR
	T_NORM_FAK : LREAL;
	T_NORM : LREAL;
	T_REAL : LREAL;
	LRSTARTPOS : LREAL;
	LRSTARTVEL : LREAL;
	R_EDGE_ABORTFROMPOSCTRL : R_TRIG;
	F_EDGE_ABORTFROMPOSCTRL : F_TRIG;
END_VAR
END_FUNCTION_BLOCK
